// TIA Portal project "Project_farmas_1234_Before_trangsfer" (V14)

(* hardware
DEVICE "S7-1200 station_1"  S7-1200 Station
   slot 0: "Rack_0"  S7-1200 Rack  Rack  V1.0
   slot 1: "PLC_1"  CPU 1215C DC/DC/DC  6ES7 215-1AG40-0XB0  V4.2
   slot 2: "DI 8x24VDC/DQ 8xRelay_1"  SM 1223 DI8/DQ8 x relay  6ES7 223-1PH32-0XB0  V2.0
DEVICE "GSD device_1"  GSD.Device.PN
   slot 0: "Rack"  Rack  V1.0
   slot 0: "Input Universal Full"  Input Universal Full
   slot 0: "Output Universal Full"  Output Universal Full
   slot 0: "multicontrol11"  MultiControl PROFINET  1101834  2.??
      slot 0: "MultiControl DAP"  MultiControl DAP
      slot 1: "PROFINET Network Interface"  PROFINET Network Interface
         slot 1: "Port 1"  Port 1
         slot 2: "Port 2"  Port 2
      slot 1: "Process Image Input_1"  Process Image Input
      slot 2: "Access Point for acyclic Services_1"  Access Point for acyclic Services
         slot 0: "Access Point for acyclic Services"  Access Point for acyclic Services
      slot 3: "Process Image Output_1"  Process Image Output
DEVICE "GSD device_2"  GSD.Device.PN
   slot 0: "Rack"  Rack  V1.0
   slot 0: "Input Universal Full"  Input Universal Full
   slot 0: "Output Universal Full"  Output Universal Full
   slot 0: "multicontrol12"  MultiControl PROFINET  1101834  2.??
      slot 0: "MultiControl DAP"  MultiControl DAP
      slot 1: "PROFINET Network Interface"  PROFINET Network Interface
         slot 1: "Port 1"  Port 1
         slot 2: "Port 2"  Port 2
      slot 1: "Process Image Input_1"  Process Image Input
      slot 2: "Access Point for acyclic Services_1"  Access Point for acyclic Services
         slot 0: "Access Point for acyclic Services"  Access Point for acyclic Services
      slot 3: "Process Image Output_1"  Process Image Output
DEVICE "GSD device_3"  GSD.Device.PN
   slot 0: "Rack"  Rack  V1.0
   slot 0: "Input Universal Full"  Input Universal Full
   slot 0: "Output Universal Full"  Output Universal Full
   slot 0: "multicontrol13"  MultiControl PROFINET  1101834  2.??
      slot 0: "MultiControl DAP"  MultiControl DAP
      slot 1: "PROFINET Network Interface"  PROFINET Network Interface
         slot 1: "Port 1"  Port 1
         slot 2: "Port 2"  Port 2
      slot 1: "Process Image Input_1"  Process Image Input
      slot 2: "Access Point for acyclic Services_1"  Access Point for acyclic Services
         slot 0: "Access Point for acyclic Services"  Access Point for acyclic Services
      slot 3: "Process Image Output_1"  Process Image Output
DEVICE "GSD device_4"  GSD.Device.PN
   slot 0: "Rack"  Rack  V1.0
   slot 0: "Input Universal Full"  Input Universal Full
   slot 0: "Output Universal Full"  Output Universal Full
   slot 0: "multicontrol14"  MultiControl PROFINET  1101834  2.??
      slot 0: "MultiControl DAP"  MultiControl DAP
      slot 1: "PROFINET Network Interface"  PROFINET Network Interface
         slot 1: "Port 1"  Port 1
         slot 2: "Port 2"  Port 2
      slot 1: "Process Image Input_1"  Process Image Input
      slot 2: "Access Point for acyclic Services_1"  Access Point for acyclic Services
         slot 0: "Access Point for acyclic Services"  Access Point for acyclic Services
      slot 3: "Process Image Output_1"  Process Image Output
DEVICE "GSD device_5"  GSD.Device.PN
   slot 0: "Rack"  Rack  V1.0
   slot 0: "Input Universal Full"  Input Universal Full
   slot 0: "Output Universal Full"  Output Universal Full
   slot 0: "multicontrol15"  MultiControl PROFINET  1101834  2.??
      slot 0: "MultiControl DAP"  MultiControl DAP
      slot 1: "PROFINET Network Interface"  PROFINET Network Interface
         slot 1: "Port 1"  Port 1
         slot 2: "Port 2"  Port 2
      slot 1: "Process Image Input_1"  Process Image Input
      slot 2: "Access Point for acyclic Services_1"  Access Point for acyclic Services
         slot 0: "Access Point for acyclic Services"  Access Point for acyclic Services
      slot 3: "Process Image Output_1"  Process Image Output
DEVICE "GSD device_6"  GSD.Device.PN
   slot 0: "Rack"  Rack  V1.0
   slot 0: "Input Universal Full"  Input Universal Full
   slot 0: "Output Universal Full"  Output Universal Full
   slot 0: "multicontrol16"  MultiControl PROFINET  1101834  2.??
      slot 0: "MultiControl DAP"  MultiControl DAP
      slot 1: "PROFINET Network Interface"  PROFINET Network Interface
         slot 1: "Port 1"  Port 1
         slot 2: "Port 2"  Port 2
      slot 1: "Process Image Input_1"  Process Image Input
      slot 2: "Access Point for acyclic Services_1"  Access Point for acyclic Services
         slot 0: "Access Point for acyclic Services"  Access Point for acyclic Services
      slot 3: "Process Image Output_1"  Process Image Output
*)

// ===== PLC "PLC_1"  CPU 1215C DC/DC/DC =====

VAR_GLOBAL   // PLC tag table "Default tag table"
   "sensor_long_transfer" AT %I0.1 : Bool;
   "sensor_home_short_transfer" AT %I0.2 : Bool;
   "sensor_start_short_transfer" AT %I0.3 : Bool;
   "sensor_1_metal_pusher" AT %I0.6 : Bool;
   "sensor_2_metal_pusher" AT %I0.5 : Bool;
   "sensor_1_scale_pusher" AT %I1.0 : Bool;
   "sensor_2_scale_pusher" AT %I0.7 : Bool;
   "sensor_drive_control" AT %I2.0 : Bool;
   "start" AT %I0.4 : Bool;
   "sensor_5_13" AT %I2.1 : Bool;
   "13_sensor_1" AT %I140.0 : Bool;
   "13_sensor_2" AT %I140.1 : Bool;
   "13_sensor_3" AT %I140.2 : Bool;
   "13_sensor_4" AT %I140.3 : Bool;
   "14_sensor_1" AT %I176.0 : Bool;
   "14_sensor_2" AT %I176.1 : Bool;
   "14_sensor_3" AT %I176.2 : Bool;
   "14_sensor_4" AT %I176.3 : Bool;
   "15_sensor_1" AT %I212.0 : Bool;
   "15_sensor_2" AT %I212.1 : Bool;
   "15_sensor_3" AT %I212.2 : Bool;
   "15_sensor_4" AT %I212.3 : Bool;
   "16_sensor_1" AT %I248.0 : Bool;
   "16_sensor_2" AT %I248.1 : Bool;
   "16_sensor_3" AT %I248.2 : Bool;
   "16_sensor_4" AT %I248.3 : Bool;
   "signal_left" AT %I1.2 : Bool;
   "signal_right" AT %I1.3 : Bool;
   "signal_reject_scale" AT %I1.5 : Bool;
   "signal_good_bad" AT %I2.3 : Bool;
   "signal_reject_metal" AT %I1.1 : Bool;
   "signal_scale" AT %I2.2 : Bool;
   "Tag_12" AT %I1.4 : Bool;
   "Tag_134" AT %I2.5 : Bool;
   "Tag_174" AT %I2.4 : Bool;
   "Tag_227" AT %I2.7 : Bool;
   "Tag_228" AT %I2.6 : Bool;
   "Tag_274" AT %I0.0 : Bool;
   "pulse_step" AT %Q0.0 : Bool;
   "direction_step" AT %Q0.1 : Bool;
   "run_left_short_transfer" AT %Q0.3 : Bool;
   "run_right_short_transfer" AT %Q0.2 : Bool;
   "run_long_transfer" AT %Q0.4 : Bool;
   "valve_metal_pusher" AT %Q0.5 : Bool;
   "valve_scale_pusher" AT %Q0.6 : Bool;
   "valve_long_transfer" AT %Q0.7 : Bool;
   "speed_drive_control" AT %Q1.0 : Bool;
   "direction_drive_control" AT %Q1.1 : Bool;
   "run_lamp" AT %Q2.0 : Bool;
   "13_RD1" AT %QB89 : Byte;
   "13_RD2" AT %QB90 : Byte;
   "13_RD3" AT %QB91 : Byte;
   "13_RD4" AT %QB92 : Byte;
   "14_RD1" AT %QB99 : Byte;
   "14_RD2" AT %QB100 : Byte;
   "14_RD3" AT %QB101 : Byte;
   "14_RD4" AT %QB102 : Byte;
   "15_RD1" AT %QB109 : Byte;
   "15_RD3" AT %QB110 : Byte;
   "15_RD2" AT %QB111 : Byte;
   "15_RD4" AT %QB112 : Byte;
   "16_RD1" AT %QB119 : Byte;
   "16_RD2" AT %QB120 : Byte;
   "16_RD3" AT %QB121 : Byte;
   "16_RD4" AT %QB122 : Byte;
   "Tag_206" AT %Q2.4 : Bool;
   "Tag_223" AT %Q2.1 : Bool;
   "Tag_224" AT %Q2.2 : Bool;
   "Tag_225" AT %Q2.3 : Bool;
   "temp_left" AT %M0.0 : Bool;
   "temp_right" AT %M0.1 : Bool;
   "temp_up_down_short_transfer" AT %M0.2 : Bool;
   "temp_stop_long_transfer" AT %M0.3 : Bool;
   "temp_metal_pusher" AT %M1.1 : Bool;
   "temp_13_sensor_1" AT %M13.1 : Bool;
   "temp_13_sensor_2" AT %M13.2 : Bool;
   "temp_13_sensor_3" AT %M13.3 : Bool;
   "temp_13_sensor_4" AT %M13.4 : Bool;
   "temp_14_sensor_1" AT %M14.1 : Bool;
   "temp_14_sensor_2" AT %M14.2 : Bool;
   "temp_14_sensor_3" AT %M14.3 : Bool;
   "temp_14_sensor_4" AT %M14.4 : Bool;
   "temp_15_sensor_1" AT %M15.1 : Bool;
   "temp_15_sensor_2" AT %M15.2 : Bool;
   "temp_15_sensor_3" AT %M15.3 : Bool;
   "temp_15_sensor_4" AT %M15.4 : Bool;
   "temp_16_sensor_1" AT %M16.1 : Bool;
   "temp_16_sensor_2" AT %M16.2 : Bool;
   "temp_16_sensor_3" AT %M16.3 : Bool;
   "temp_16_sensor_4" AT %M16.4 : Bool;
   "temp_drive_control" AT %M17.0 : Bool;
   "temp_signal_good_bad" AT %M17.1 : Bool;
   "temp_reject_metal" AT %M17.2 : Bool;
   "temp_reject_scale" AT %M17.3 : Bool;
   "temp_scale_pusher" AT %M1.2 : Bool;
   "Tag_1" AT %M16.6 : Bool;
   "Tag_2" AT %M0.4 : Bool;
   "Tag_3" AT %M100.0 : Bool;
   "Tag_4" AT %M100.1 : Bool;
   "Tag_5" AT %M100.2 : Bool;
   "Tag_6" AT %M100.3 : Bool;
   "Tag_7" AT %M100.4 : Bool;
   "Tag_8" AT %M100.6 : Bool;
   "Tag_9" AT %M101.0 : Bool;
   "Tag_10" AT %M101.5 : Bool;
   "Tag_11" AT %M105.6 : Bool;
   "Tag_13" AT %M150.0 : Bool;
   "Tag_14" AT %M150.1 : Bool;
   "Tag_15" AT %M200.2 : Bool;
   "Tag_16" AT %M1000.0 : Bool;
   "Tag_17" AT %M200.1 : Bool;
   "Tag_18" AT %M1000.1 : Bool;
   "Tag_19" AT %M1000.2 : Bool;
   "Tag_20" AT %M200.7 : Bool;
   "Tag_21" AT %M200.0 : Bool;
   "Tag_22" AT %M201.1 : Bool;
   "Tag_23" AT %M151.0 : Bool;
   "Tag_24" AT %M151.1 : Bool;
   "Tag_25" AT %M201.7 : Bool;
   "Tag_26" AT %M149.0 : Bool;
   "Tag_27" AT %M149.1 : Bool;
   "Tag_28" AT %M199.7 : Bool;
   "Tag_29" AT %M199.0 : Bool;
   "Tag_30" AT %M199.1 : Bool;
   "Tag_31" AT %M999.0 : Bool;
   "Tag_32" AT %M999.1 : Bool;
   "Tag_33" AT %M999.2 : Bool;
   "Tag_34" AT %M199.2 : Bool;
   "Tag_35" AT %M202.1 : Bool;
   "Tag_36" AT %M201.0 : Bool;
   "Tag_37" AT %M201.2 : Bool;
   "Tag_38" AT %M1001.2 : Bool;
   "Tag_39" AT %M1001.1 : Bool;
   "Tag_40" AT %M1001.0 : Bool;
   "Tag_41" AT %M158.0 : Bool;
   "Tag_42" AT %M158.1 : Bool;
   "Tag_43" AT %M208.7 : Bool;
   "Tag_44" AT %M203.1 : Bool;
   "Tag_45" AT %M208.0 : Bool;
   "Tag_46" AT %M208.1 : Bool;
   "Tag_47" AT %M159.0 : Bool;
   "Tag_48" AT %M159.1 : Bool;
   "Tag_49" AT %M209.7 : Bool;
   "Tag_50" AT %M210.1 : Bool;
   "Tag_51" AT %M209.0 : Bool;
   "Tag_52" AT %M209.1 : Bool;
   "Tag_53" AT %M209.2 : Bool;
   "Tag_54" AT %M1009.0 : Bool;
   "Tag_55" AT %M1009.1 : Bool;
   "Tag_56" AT %M160.0 : Bool;
   "Tag_57" AT %M160.1 : Bool;
   "Tag_58" AT %M210.7 : Bool;
   "Tag_59" AT %M211.1 : Bool;
   "Tag_60" AT %M210.0 : Bool;
   "Tag_61" AT %M210.2 : Bool;
   "Tag_62" AT %M161.0 : Bool;
   "Tag_63" AT %M161.1 : Bool;
   "Tag_64" AT %M211.7 : Bool;
   "Tag_65" AT %M212.1 : Bool;
   "Tag_66" AT %M211.0 : Bool;
   "Tag_67" AT %M1010.0 : Bool;
   "Tag_68" AT %M1010.1 : Bool;
   "Tag_69" AT %M1010.2 : Bool;
   "Tag_70" AT %M211.2 : Bool;
   "Tag_71" AT %M1011.0 : Bool;
   "Tag_72" AT %M1011.1 : Bool;
   "Tag_73" AT %M1011.2 : Bool;
   "Tag_74" AT %M162.0 : Bool;
   "Tag_75" AT %M162.1 : Bool;
   "Tag_76" AT %M212.7 : Bool;
   "Tag_77" AT %M213.1 : Bool;
   "Tag_78" AT %M212.0 : Bool;
   "Tag_79" AT %M153.0 : Bool;
   "Tag_80" AT %M153.1 : Bool;
   "Tag_81" AT %M156.0 : Bool;
   "Tag_82" AT %M156.1 : Bool;
   "Tag_83" AT %M206.7 : Bool;
   "Tag_84" AT %M206.0 : Bool;
   "Tag_85" AT %M206.1 : Bool;
   "Tag_86" AT %M206.2 : Bool;
   "Tag_87" AT %M1006.0 : Bool;
   "Tag_88" AT %M1006.1 : Bool;
   "Tag_89" AT %M1006.2 : Bool;
   "Tag_90" AT %M152.0 : Bool;
   "Tag_91" AT %M152.1 : Bool;
   "Tag_92" AT %M202.7 : Bool;
   "Tag_93" AT %M202.0 : Bool;
   "Tag_94" AT %M202.2 : Bool;
   "Tag_95" AT %M203.3 : Bool;
   "Tag_96" AT %M1002.0 : Bool;
   "Tag_97" AT %M1002.1 : Bool;
   "Tag_98" AT %M1002.2 : Bool;
   "Tag_99" AT %M207.5 : Bool;
   "Tag_100" AT %M203.7 : Bool;
   "Tag_101" AT %M204.1 : Bool;
   "Tag_102" AT %M203.0 : Bool;
   "Tag_103" AT %M203.2 : Bool;
   "Tag_104" AT %M1003.2 : Bool;
   "Tag_105" AT %M203.4 : Bool;
   "Tag_106" AT %M204.5 : Bool;
   "Tag_107" AT %M1006.5 : Bool;
   "Tag_108" AT %M207.4 : Bool;
   "Tag_109" AT %M1006.6 : Bool;
   "Tag_110" AT %M1007.0 : Bool;
   "Tag_111" AT %M1007.1 : Bool;
   "Tag_112" AT %M1007.2 : Bool;
   "Tag_113" AT %M1007.4 : Bool;
   "Tag_114" AT %M1007.5 : Bool;
   "Tag_115" AT %M208.2 : Bool;
   "Tag_116" AT %M1008.0 : Bool;
   "Tag_117" AT %M1008.1 : Bool;
   "Tag_118" AT %M1008.2 : Bool;
   "Tag_119" AT %M147.0 : Bool;
   "Tag_120" AT %M1008.6 : Bool;
   "Tag_121" AT %M1008.7 : Bool;
   "Tag_122" AT %M198.0 : Bool;
   "Tag_123" AT %M300.7 : Bool;
   "Tag_124" AT %M212.2 : Bool;
   "Tag_125" AT %M1012.0 : Bool;
   "Tag_126" AT %M1012.1 : Bool;
   "Tag_127" AT %M1012.2 : Bool;
   "Tag_128" AT %M163.0 : Bool;
   "Tag_129" AT %M163.1 : Bool;
   "Tag_130" AT %M213.7 : Bool;
   "Tag_131" AT %M214.1 : Bool;
   "Tag_132" AT %M213.0 : Bool;
   "Tag_133" AT %M213.2 : Bool;
   "Tag_135" AT %M1001.3 : Bool;
   "Tag_136" AT %M1013.0 : Bool;
   "Tag_137" AT %M1013.3 : Bool;
   "Tag_138" AT %M1013.1 : Bool;
   "Tag_139" AT %M1013.2 : Bool;
   "Tag_140" AT %M164.0 : Bool;
   "Tag_141" AT %M164.1 : Bool;
   "Tag_142" AT %M214.7 : Bool;
   "Tag_143" AT %M215.1 : Bool;
   "Tag_144" AT %M214.0 : Bool;
   "Tag_145" AT %M217.0 : Bool;
   "Tag_146" AT %M214.2 : Bool;
   "Tag_147" AT %M1014.0 : Bool;
   "Tag_148" AT %M1014.1 : Bool;
   "Tag_149" AT %M1014.2 : Bool;
   "Tag_150" AT %M0.5 : Bool;
   "Tag_151" AT %M1020.0 : Bool;
   "Tag_152" AT %M1020.7 : Bool;
   "Tag_153" AT %M1021.0 : Bool;
   "Tag_154" AT %M1021.1 : Bool;
   "Tag_155" AT %M1022.2 : Bool;
   "Tag_156" AT %M146.1 : Bool;
   "Tag_157" AT %M146.0 : Bool;
   "Tag_158" AT %M1023.0 : Bool;
   "Tag_159" AT %M165.0 : Bool;
   "Tag_160" AT %M165.1 : Bool;
   "Tag_161" AT %M215.7 : Bool;
   "Tag_162" AT %M216.1 : Bool;
   "Tag_163" AT %M215.0 : Bool;
   "Tag_164" AT %M215.2 : Bool;
   "Tag_165" AT %M1015.0 : Bool;
   "Tag_166" AT %M214.3 : Bool;
   "Tag_167" AT %M1025.0 : Bool;
   "Tag_168" AT %M1025.1 : Bool;
   "Tag_169" AT %M166.0 : Bool;
   "Tag_170" AT %M166.1 : Bool;
   "Tag_171" AT %M216.7 : Bool;
   "Tag_172" AT %M217.1 : Bool;
   "Tag_173" AT %M216.0 : Bool;
   "Tag_175" AT %M216.2 : Bool;
   "Tag_176" AT %M1016.0 : Bool;
   "Tag_177" AT %M1016.1 : Bool;
   "Tag_178" AT %M1016.2 : Bool;
   "Tag_179" AT %MW10 : Word;
   "Tag_180" AT %M1023.2 : Bool;
   "Tag_181" AT %M1023.3 : Bool;
   "Tag_182" AT %M1024.0 : Bool;
   "Tag_183" AT %M1024.1 : Bool;
   "Tag_184" AT %M1024.4 : Bool;
   "Tag_185" AT %M170.0 : Bool;
   "System_Byte" AT %MB4095 : Byte;
   "FirstScan" AT %M4095.0 : Bool;
   "DiagStatusUpdate" AT %M4095.1 : Bool;
   "AlwaysTRUE" AT %M4095.2 : Bool;
   "AlwaysFALSE" AT %M4095.3 : Bool;
   "System_Byte(1)" AT %MB1 : Byte;
   "Tag_186" AT %M1026.4 : Bool;
   "Tag_187" AT %M1028.0 : Bool;
   "Tag_188" AT %M1027.0 : Bool;
   "Tag_189" AT %M1500.0 : Bool;
   "Tag_190" AT %M208.5 : Bool;
   "Tag_191" AT %M1036.5 : Bool;
   "Tag_192" AT %M1030.0 : Bool;
   "Tag_193" AT %M1030.1 : Bool;
   "Tag_194" AT %M1035.2 : Bool;
   "Tag_195" AT %M1035.3 : Bool;
   "Tag_196" AT %M1035.6 : Bool;
   "Tag_197" AT %M1036.0 : Bool;
   "Tag_198" AT %M1033.6 : Bool;
   "Tag_199" AT %M300.3 : Bool;
   "Tag_200" AT %M1044.0 : Bool;
   "Tag_201" AT %M300.2 : Bool;
   "Tag_202" AT %M1044.1 : Bool;
   "Tag_203" AT %M1040.0 : Bool;
   "Tag_204" AT %M1040.3 : Bool;
   "Tag_205" AT %M1047.0 : Bool;
   "Tag_207" AT %M400.0 : Bool;
   "Tag_208" AT %M400.1 : Bool;
   "Tag_209" AT %M399.0 : Bool;
   "Tag_210" AT %M400.5 : Bool;
   "Tag_211" AT %M400.6 : Bool;
   "Tag_212" AT %M400.7 : Bool;
   "Tag_213" AT %M800.0 : Bool;
   "Tag_214" AT %M800.3 : Bool;
   "Tag_215" AT %M801.0 : Bool;
   "Tag_216" AT %M401.1 : Bool;
   "Tag_217" AT %M801.1 : Bool;
   "Tag_218" AT %M401.2 : Bool;
   "Tag_219" AT %M801.2 : Bool;
   "Tag_220" AT %M1080.0 : Bool;
   "Tag_221" AT %M404.0 : Bool;
   "Tag_222" AT %M500.0 : Bool;
   "Tag_226" AT %M500.1 : Bool;
   "Clock_Byte" AT %MB410 : Byte;
   "Clock_10Hz" AT %M410.0 : Bool;
   "Clock_5Hz" AT %M410.1 : Bool;
   "Clock_2.5Hz" AT %M410.2 : Bool;
   "Clock_2Hz" AT %M410.3 : Bool;
   "Clock_1.25Hz" AT %M410.4 : Bool;
   "Clock_1Hz" AT %M410.5 : Bool;
   "Clock_0.625Hz" AT %M410.6 : Bool;
   "Clock_0.5Hz" AT %M410.7 : Bool;
   "Tag_229" AT %M420.0 : Bool;
   "Tag_230" AT %M500.2 : Bool;
   "Tag_231" AT %M420.1 : Bool;
   "Tag_232" AT %M500.3 : Bool;
   "Tag_233" AT %M500.4 : Bool;
   "Tag_234" AT %M400.4 : Bool;
   "Tag_235" AT %M420.4 : Bool;
   "Tag_236" AT %M500.7 : Bool;
   "Tag_237" AT %M1053.0 : Bool;
   "Tag_238" AT %M1053.1 : Bool;
   "Tag_239" AT %M1053.3 : Bool;
   "Tag_240" AT %M1070.0 : Bool;
   "Tag_241" AT %M700.0 : Bool;
   "Tag_242" AT %M489.0 : Bool;
   "Tag_243" AT %M500.5 : Bool;
   "Tag_244" AT %M500.6 : Bool;
   "Tag_245" AT %M1071.1 : Bool;
   "Tag_246" AT %M293.1 : Bool;
   "Tag_247" AT %M1071.2 : Bool;
   "Tag_248" AT %M1071.3 : Bool;
   "Tag_249" AT %M1071.4 : Bool;
   "Tag_250" AT %M1072.1 : Bool;
   "Tag_251" AT %M293.2 : Bool;
   "Tag_252" AT %M388.0 : Bool;
   "Tag_253" AT %M1077.2 : Bool;
   "Tag_254" AT %M2.6 : Bool;
   "Tag_255" AT %M1074.0 : Bool;
   "Tag_256" AT %M1075.0 : Bool;
   "Tag_257" AT %M183.0 : Bool;
   "Tag_258" AT %M1090.0 : Bool;
   "Tag_259" AT %M1090.1 : Bool;
   "Tag_260" AT %M1090.3 : Bool;
   "Tag_261" AT %M1090.4 : Bool;
   "Tag_262" AT %M1090.5 : Bool;
   "Tag_263" AT %M1090.6 : Bool;
   "Tag_264" AT %M1091.0 : Bool;
   "Tag_265" AT %M1091.1 : Bool;
   "Tag_266" AT %M1060.0 : Bool;
   "Tag_267" AT %M1060.1 : Bool;
   "Tag_268" AT %M1060.2 : Bool;
   "Tag_269" AT %M1060.3 : Bool;
   "Tag_270" AT %M1060.4 : Bool;
   "Tag_271" AT %M1060.5 : Bool;
   "Tag_272" AT %M1060.6 : Bool;
   "Tag_273" AT %M489.1 : Bool;
   "Tag_275" AT %M1061.0 : Bool;
   "Tag_276" AT %M489.2 : Bool;
   "Tag_277" AT %M489.4 : Bool;
   "Tag_278" AT %M1061.2 : Bool;
END_VAR

DATA_BLOCK "Connect_PC"   // DB1
{ S7_Optimized_Access := 'FALSE' }
VERSION : 0.1
   VAR
      Scan_check_metal : Byte := 0;
      weight_pusher : Byte := 0;
      print_pusher : Byte := 0;
      sensor_before_metal_scan : Byte := 0;
      metal_check_result : Byte := 0;
      sensor_after_metal_check : Byte := 0;
      metal_pusher : Byte := 0;
      sensor_tranfer : Byte := 0;
      sensor_left : Byte := 0;
      sensor_right : Byte := 0;
      EMG : Byte := 0;
   END_VAR
BEGIN
END_DATA_BLOCK

// folder: System blocks/Program resources

DATA_BLOCK "TZ7-1"   // DB6
{ S7_Optimized_Access := 'TRUE' }
AUTHOR : Simatic
FAMILY : IEC
NAME : IEC_TMR
VERSION : 1.0
// stored: InstanceOfName IEC_TIMER
"IEC_TIMER"
BEGIN
END_DATA_BLOCK

DATA_BLOCK "IEC_Timer_0_DB"   // DB7
{ S7_Optimized_Access := 'TRUE' }
AUTHOR : Simatic
FAMILY : IEC
NAME : IEC_TMR
VERSION : 1.0
// stored: InstanceOfName IEC_TIMER
"IEC_TIMER"
BEGIN
END_DATA_BLOCK

DATA_BLOCK "T13-1"   // DB8
{ S7_Optimized_Access := 'TRUE' }
AUTHOR : Simatic
FAMILY : IEC
NAME : IEC_TMR
VERSION : 1.0
// stored: InstanceOfName IEC_TIMER
"IEC_TIMER"
BEGIN
END_DATA_BLOCK

DATA_BLOCK "T13-2"   // DB9
{ S7_Optimized_Access := 'TRUE' }
AUTHOR : Simatic
FAMILY : IEC
NAME : IEC_TMR
VERSION : 1.0
// stored: InstanceOfName IEC_TIMER
"IEC_TIMER"
BEGIN
END_DATA_BLOCK

DATA_BLOCK "IEC_Timer_0_DB_9"   // DB10
{ S7_Optimized_Access := 'TRUE' }
AUTHOR : Simatic
FAMILY : IEC
NAME : IEC_TMR
VERSION : 1.0
// stored: InstanceOfName IEC_TIMER
"IEC_TIMER"
BEGIN
END_DATA_BLOCK

DATA_BLOCK "T9-1"   // DB11
{ S7_Optimized_Access := 'TRUE' }
AUTHOR : Simatic
FAMILY : IEC
NAME : IEC_TMR
VERSION : 1.0
// stored: InstanceOfName IEC_TIMER
"IEC_TIMER"
BEGIN
END_DATA_BLOCK

DATA_BLOCK "IEC_Timer_0_DB_1"   // DB12
{ S7_Optimized_Access := 'TRUE' }
AUTHOR : Simatic
FAMILY : IEC
NAME : IEC_TMR
VERSION : 1.0
// stored: InstanceOfName IEC_TIMER
"IEC_TIMER"
BEGIN
END_DATA_BLOCK

DATA_BLOCK "IEC_Timer_0_DB_2"   // DB13
{ S7_Optimized_Access := 'TRUE' }
AUTHOR : Simatic
FAMILY : IEC
NAME : IEC_TMR
VERSION : 1.0
// stored: InstanceOfName IEC_TIMER
"IEC_TIMER"
BEGIN
END_DATA_BLOCK

DATA_BLOCK "IEC_Timer_0_DB_3"   // DB14
{ S7_Optimized_Access := 'TRUE' }
AUTHOR : Simatic
FAMILY : IEC
NAME : IEC_TMR
VERSION : 1.0
// stored: InstanceOfName IEC_TIMER
"IEC_TIMER"
BEGIN
END_DATA_BLOCK

DATA_BLOCK "IEC_Timer_0_DB_4"   // DB15
{ S7_Optimized_Access := 'TRUE' }
AUTHOR : Simatic
FAMILY : IEC
NAME : IEC_TMR
VERSION : 1.0
// stored: InstanceOfName IEC_TIMER
"IEC_TIMER"
BEGIN
END_DATA_BLOCK

DATA_BLOCK "TZ12-1"   // DB16
{ S7_Optimized_Access := 'TRUE' }
AUTHOR : Simatic
FAMILY : IEC
NAME : IEC_TMR
VERSION : 1.0
// stored: InstanceOfName IEC_TIMER
"IEC_TIMER"
BEGIN
END_DATA_BLOCK

DATA_BLOCK "T3-1"   // DB17
{ S7_Optimized_Access := 'TRUE' }
AUTHOR : Simatic
FAMILY : IEC
NAME : IEC_TMR
VERSION : 1.0
// stored: InstanceOfName IEC_TIMER
"IEC_TIMER"
BEGIN
END_DATA_BLOCK

DATA_BLOCK "TZ3-1"   // DB18
{ S7_Optimized_Access := 'TRUE' }
AUTHOR : Simatic
FAMILY : IEC
NAME : IEC_TMR
VERSION : 1.0
// stored: InstanceOfName IEC_TIMER
"IEC_TIMER"
BEGIN
END_DATA_BLOCK

DATA_BLOCK "TZ3-2"   // DB19
{ S7_Optimized_Access := 'TRUE' }
AUTHOR : Simatic
FAMILY : IEC
NAME : IEC_TMR
VERSION : 1.0
// stored: InstanceOfName IEC_TIMER
"IEC_TIMER"
BEGIN
END_DATA_BLOCK

DATA_BLOCK "TZ5-2"   // DB20
{ S7_Optimized_Access := 'TRUE' }
AUTHOR : Simatic
FAMILY : IEC
NAME : IEC_TMR
VERSION : 1.0
// stored: InstanceOfName IEC_TIMER
"IEC_TIMER"
BEGIN
END_DATA_BLOCK

DATA_BLOCK "TZ5-1"   // DB21
{ S7_Optimized_Access := 'TRUE' }
AUTHOR : Simatic
FAMILY : IEC
NAME : IEC_TMR
VERSION : 1.0
// stored: InstanceOfName IEC_TIMER
"IEC_TIMER"
BEGIN
END_DATA_BLOCK

DATA_BLOCK "T5-1"   // DB22
{ S7_Optimized_Access := 'TRUE' }
AUTHOR : Simatic
FAMILY : IEC
NAME : IEC_TMR
VERSION : 1.0
// stored: InstanceOfName IEC_TIMER
"IEC_TIMER"
BEGIN
END_DATA_BLOCK

DATA_BLOCK "T5-2"   // DB23
{ S7_Optimized_Access := 'TRUE' }
AUTHOR : Simatic
FAMILY : IEC
NAME : IEC_TMR
VERSION : 1.0
// stored: InstanceOfName IEC_TIMER
"IEC_TIMER"
BEGIN
END_DATA_BLOCK

DATA_BLOCK "T9-2"   // DB24
{ S7_Optimized_Access := 'TRUE' }
AUTHOR : Simatic
FAMILY : IEC
NAME : IEC_TMR
VERSION : 1.0
// stored: InstanceOfName IEC_TIMER
"IEC_TIMER"
BEGIN
END_DATA_BLOCK

DATA_BLOCK "T10-1"   // DB25
{ S7_Optimized_Access := 'TRUE' }
AUTHOR : Simatic
FAMILY : IEC
NAME : IEC_TMR
VERSION : 1.0
// stored: InstanceOfName IEC_TIMER
"IEC_TIMER"
BEGIN
END_DATA_BLOCK

DATA_BLOCK "T10-2"   // DB26
{ S7_Optimized_Access := 'TRUE' }
AUTHOR : Simatic
FAMILY : IEC
NAME : IEC_TMR
VERSION : 1.0
// stored: InstanceOfName IEC_TIMER
"IEC_TIMER"
BEGIN
END_DATA_BLOCK

DATA_BLOCK "TZ10-1"   // DB27
{ S7_Optimized_Access := 'TRUE' }
AUTHOR : Simatic
FAMILY : IEC
NAME : IEC_TMR
VERSION : 1.0
// stored: InstanceOfName IEC_TIMER
"IEC_TIMER"
BEGIN
END_DATA_BLOCK

DATA_BLOCK "TZ10-2"   // DB28
{ S7_Optimized_Access := 'TRUE' }
AUTHOR : Simatic
FAMILY : IEC
NAME : IEC_TMR
VERSION : 1.0
// stored: InstanceOfName IEC_TIMER
"IEC_TIMER"
BEGIN
END_DATA_BLOCK

DATA_BLOCK "TZ9-2"   // DB29
{ S7_Optimized_Access := 'TRUE' }
AUTHOR : Simatic
FAMILY : IEC
NAME : IEC_TMR
VERSION : 1.0
// stored: InstanceOfName IEC_TIMER
"IEC_TIMER"
BEGIN
END_DATA_BLOCK

DATA_BLOCK "TZ9-1"   // DB30
{ S7_Optimized_Access := 'TRUE' }
AUTHOR : Simatic
FAMILY : IEC
NAME : IEC_TMR
VERSION : 1.0
// stored: InstanceOfName IEC_TIMER
"IEC_TIMER"
BEGIN
END_DATA_BLOCK

DATA_BLOCK "TZ11-2"   // DB31
{ S7_Optimized_Access := 'TRUE' }
AUTHOR : Simatic
FAMILY : IEC
NAME : IEC_TMR
VERSION : 1.0
// stored: InstanceOfName IEC_TIMER
"IEC_TIMER"
BEGIN
END_DATA_BLOCK

DATA_BLOCK "TZ11-1"   // DB32
{ S7_Optimized_Access := 'TRUE' }
AUTHOR : Simatic
FAMILY : IEC
NAME : IEC_TMR
VERSION : 1.0
// stored: InstanceOfName IEC_TIMER
"IEC_TIMER"
BEGIN
END_DATA_BLOCK

DATA_BLOCK "T11-1"   // DB33
{ S7_Optimized_Access := 'TRUE' }
AUTHOR : Simatic
FAMILY : IEC
NAME : IEC_TMR
VERSION : 1.0
// stored: InstanceOfName IEC_TIMER
"IEC_TIMER"
BEGIN
END_DATA_BLOCK

DATA_BLOCK "T11-2"   // DB34
{ S7_Optimized_Access := 'TRUE' }
AUTHOR : Simatic
FAMILY : IEC
NAME : IEC_TMR
VERSION : 1.0
// stored: InstanceOfName IEC_TIMER
"IEC_TIMER"
BEGIN
END_DATA_BLOCK

DATA_BLOCK "T12-1"   // DB35
{ S7_Optimized_Access := 'TRUE' }
AUTHOR : Simatic
FAMILY : IEC
NAME : IEC_TMR
VERSION : 1.0
// stored: InstanceOfName IEC_TIMER
"IEC_TIMER"
BEGIN
END_DATA_BLOCK

DATA_BLOCK "T12-2"   // DB36
{ S7_Optimized_Access := 'TRUE' }
AUTHOR : Simatic
FAMILY : IEC
NAME : IEC_TMR
VERSION : 1.0
// stored: InstanceOfName IEC_TIMER
"IEC_TIMER"
BEGIN
END_DATA_BLOCK

DATA_BLOCK "TZ2-1"   // DB37
{ S7_Optimized_Access := 'TRUE' }
AUTHOR : Simatic
FAMILY : IEC
NAME : IEC_TMR
VERSION : 1.0
// stored: InstanceOfName IEC_TIMER
"IEC_TIMER"
BEGIN
END_DATA_BLOCK

DATA_BLOCK "TZ2-2"   // DB38
{ S7_Optimized_Access := 'TRUE' }
AUTHOR : Simatic
FAMILY : IEC
NAME : IEC_TMR
VERSION : 1.0
// stored: InstanceOfName IEC_TIMER
"IEC_TIMER"
BEGIN
END_DATA_BLOCK

DATA_BLOCK "T2-1"   // DB39
{ S7_Optimized_Access := 'TRUE' }
AUTHOR : Simatic
FAMILY : IEC
NAME : IEC_TMR
VERSION : 1.0
// stored: InstanceOfName IEC_TIMER
"IEC_TIMER"
BEGIN
END_DATA_BLOCK

DATA_BLOCK "T2-2"   // DB40
{ S7_Optimized_Access := 'TRUE' }
AUTHOR : Simatic
FAMILY : IEC
NAME : IEC_TMR
VERSION : 1.0
// stored: InstanceOfName IEC_TIMER
"IEC_TIMER"
BEGIN
END_DATA_BLOCK

DATA_BLOCK "T3-2"   // DB41
{ S7_Optimized_Access := 'TRUE' }
AUTHOR : Simatic
FAMILY : IEC
NAME : IEC_TMR
VERSION : 1.0
// stored: InstanceOfName IEC_TIMER
"IEC_TIMER"
BEGIN
END_DATA_BLOCK

DATA_BLOCK "TZ12-2"   // DB42
{ S7_Optimized_Access := 'TRUE' }
AUTHOR : Simatic
FAMILY : IEC
NAME : IEC_TMR
VERSION : 1.0
// stored: InstanceOfName IEC_TIMER
"IEC_TIMER"
BEGIN
END_DATA_BLOCK

DATA_BLOCK "T6-1"   // DB43
{ S7_Optimized_Access := 'TRUE' }
AUTHOR : Simatic
FAMILY : IEC
NAME : IEC_TMR
VERSION : 1.0
// stored: InstanceOfName IEC_TIMER
"IEC_TIMER"
BEGIN
END_DATA_BLOCK

DATA_BLOCK "TZ13-1"   // DB44
{ S7_Optimized_Access := 'TRUE' }
AUTHOR : Simatic
FAMILY : IEC
NAME : IEC_TMR
VERSION : 1.0
// stored: InstanceOfName IEC_TIMER
"IEC_TIMER"
BEGIN
END_DATA_BLOCK

DATA_BLOCK "TZ6-1"   // DB45
{ S7_Optimized_Access := 'TRUE' }
AUTHOR : Simatic
FAMILY : IEC
NAME : IEC_TMR
VERSION : 1.0
// stored: InstanceOfName IEC_TIMER
"IEC_TIMER"
BEGIN
END_DATA_BLOCK

DATA_BLOCK "TZ6-2"   // DB46
{ S7_Optimized_Access := 'TRUE' }
AUTHOR : Simatic
FAMILY : IEC
NAME : IEC_TMR
VERSION : 1.0
// stored: InstanceOfName IEC_TIMER
"IEC_TIMER"
BEGIN
END_DATA_BLOCK

DATA_BLOCK "T6-2"   // DB47
{ S7_Optimized_Access := 'TRUE' }
AUTHOR : Simatic
FAMILY : IEC
NAME : IEC_TMR
VERSION : 1.0
// stored: InstanceOfName IEC_TIMER
"IEC_TIMER"
BEGIN
END_DATA_BLOCK

DATA_BLOCK "TZ13-2"   // DB48
{ S7_Optimized_Access := 'TRUE' }
AUTHOR : Simatic
FAMILY : IEC
NAME : IEC_TMR
VERSION : 1.0
// stored: InstanceOfName IEC_TIMER
"IEC_TIMER"
BEGIN
END_DATA_BLOCK

DATA_BLOCK "T-metal"   // DB49
{ S7_Optimized_Access := 'TRUE' }
AUTHOR : Simatic
FAMILY : IEC
NAME : IEC_TMR
VERSION : 1.0
// stored: InstanceOfName IEC_TIMER
"IEC_TIMER"
BEGIN
END_DATA_BLOCK

DATA_BLOCK "T7-2"   // DB50
{ S7_Optimized_Access := 'TRUE' }
AUTHOR : Simatic
FAMILY : IEC
NAME : IEC_TMR
VERSION : 1.0
// stored: InstanceOfName IEC_TIMER
"IEC_TIMER"
BEGIN
END_DATA_BLOCK

DATA_BLOCK "TZ7-2"   // DB51
{ S7_Optimized_Access := 'TRUE' }
AUTHOR : Simatic
FAMILY : IEC
NAME : IEC_TMR
VERSION : 1.0
// stored: InstanceOfName IEC_TIMER
"IEC_TIMER"
BEGIN
END_DATA_BLOCK

DATA_BLOCK "TZ7-3"   // DB52
{ S7_Optimized_Access := 'TRUE' }
AUTHOR : Simatic
FAMILY : IEC
NAME : IEC_TMR
VERSION : 1.0
// stored: InstanceOfName IEC_TIMER
"IEC_TIMER"
BEGIN
END_DATA_BLOCK

DATA_BLOCK "TM207"   // DB53
{ S7_Optimized_Access := 'TRUE' }
AUTHOR : Simatic
FAMILY : IEC
NAME : IEC_TMR
VERSION : 1.0
// stored: InstanceOfName IEC_TIMER
"IEC_TIMER"
BEGIN
END_DATA_BLOCK

DATA_BLOCK "IEC_Timer_0_DB_5"   // DB54
{ S7_Optimized_Access := 'TRUE' }
AUTHOR : Simatic
FAMILY : IEC
NAME : IEC_TMR
VERSION : 1.0
// stored: InstanceOfName IEC_TIMER
"IEC_TIMER"
BEGIN
END_DATA_BLOCK

DATA_BLOCK "TZ8-1"   // DB55
{ S7_Optimized_Access := 'TRUE' }
AUTHOR : Simatic
FAMILY : IEC
NAME : IEC_TMR
VERSION : 1.0
// stored: InstanceOfName IEC_TIMER
"IEC_TIMER"
BEGIN
END_DATA_BLOCK

DATA_BLOCK "TZ8-2"   // DB56
{ S7_Optimized_Access := 'TRUE' }
AUTHOR : Simatic
FAMILY : IEC
NAME : IEC_TMR
VERSION : 1.0
// stored: InstanceOfName IEC_TIMER
"IEC_TIMER"
BEGIN
END_DATA_BLOCK

DATA_BLOCK "T8-1"   // DB57
{ S7_Optimized_Access := 'TRUE' }
AUTHOR : Simatic
FAMILY : IEC
NAME : IEC_TMR
VERSION : 1.0
// stored: InstanceOfName IEC_TIMER
"IEC_TIMER"
BEGIN
END_DATA_BLOCK

DATA_BLOCK "T8-2"   // DB58
{ S7_Optimized_Access := 'TRUE' }
AUTHOR : Simatic
FAMILY : IEC
NAME : IEC_TMR
VERSION : 1.0
// stored: InstanceOfName IEC_TIMER
"IEC_TIMER"
BEGIN
END_DATA_BLOCK

DATA_BLOCK "TZ14-2"   // DB59
{ S7_Optimized_Access := 'TRUE' }
AUTHOR : Simatic
FAMILY : IEC
NAME : IEC_TMR
VERSION : 1.0
// stored: InstanceOfName IEC_TIMER
"IEC_TIMER"
BEGIN
END_DATA_BLOCK

DATA_BLOCK "TZ14-1"   // DB60
{ S7_Optimized_Access := 'TRUE' }
AUTHOR : Simatic
FAMILY : IEC
NAME : IEC_TMR
VERSION : 1.0
// stored: InstanceOfName IEC_TIMER
"IEC_TIMER"
BEGIN
END_DATA_BLOCK

DATA_BLOCK "T14-1"   // DB61
{ S7_Optimized_Access := 'TRUE' }
AUTHOR : Simatic
FAMILY : IEC
NAME : IEC_TMR
VERSION : 1.0
// stored: InstanceOfName IEC_TIMER
"IEC_TIMER"
BEGIN
END_DATA_BLOCK

DATA_BLOCK "T14-2"   // DB62
{ S7_Optimized_Access := 'TRUE' }
AUTHOR : Simatic
FAMILY : IEC
NAME : IEC_TMR
VERSION : 1.0
// stored: InstanceOfName IEC_TIMER
"IEC_TIMER"
BEGIN
END_DATA_BLOCK

DATA_BLOCK "T-SCALE"   // DB63
{ S7_Optimized_Access := 'TRUE' }
AUTHOR : Simatic
FAMILY : IEC
NAME : IEC_TMR
VERSION : 1.0
// stored: InstanceOfName IEC_TIMER
"IEC_TIMER"
BEGIN
END_DATA_BLOCK

DATA_BLOCK "IEC_Timer_0_DB_7"   // DB64
{ S7_Optimized_Access := 'TRUE' }
AUTHOR : Simatic
FAMILY : IEC
NAME : IEC_TMR
VERSION : 1.0
// stored: InstanceOfName IEC_TIMER
"IEC_TIMER"
BEGIN
END_DATA_BLOCK

DATA_BLOCK "IEC_Timer_0_DB_8"   // DB65
{ S7_Optimized_Access := 'TRUE' }
AUTHOR : Simatic
FAMILY : IEC
NAME : IEC_TMR
VERSION : 1.0
// stored: InstanceOfName IEC_TIMER
"IEC_TIMER"
BEGIN
END_DATA_BLOCK

DATA_BLOCK "TZ15-1"   // DB66
{ S7_Optimized_Access := 'TRUE' }
AUTHOR : Simatic
FAMILY : IEC
NAME : IEC_TMR
VERSION : 1.0
// stored: InstanceOfName IEC_TIMER
"IEC_TIMER"
BEGIN
END_DATA_BLOCK

DATA_BLOCK "TZ15-2"   // DB67
{ S7_Optimized_Access := 'TRUE' }
AUTHOR : Simatic
FAMILY : IEC
NAME : IEC_TMR
VERSION : 1.0
// stored: InstanceOfName IEC_TIMER
"IEC_TIMER"
BEGIN
END_DATA_BLOCK

DATA_BLOCK "T15-1"   // DB68
{ S7_Optimized_Access := 'TRUE' }
AUTHOR : Simatic
FAMILY : IEC
NAME : IEC_TMR
VERSION : 1.0
// stored: InstanceOfName IEC_TIMER
"IEC_TIMER"
BEGIN
END_DATA_BLOCK

DATA_BLOCK "T15-2"   // DB69
{ S7_Optimized_Access := 'TRUE' }
AUTHOR : Simatic
FAMILY : IEC
NAME : IEC_TMR
VERSION : 1.0
// stored: InstanceOfName IEC_TIMER
"IEC_TIMER"
BEGIN
END_DATA_BLOCK

DATA_BLOCK "T16-1"   // DB70
{ S7_Optimized_Access := 'TRUE' }
AUTHOR : Simatic
FAMILY : IEC
NAME : IEC_TMR
VERSION : 1.0
// stored: InstanceOfName IEC_TIMER
"IEC_TIMER"
BEGIN
END_DATA_BLOCK

DATA_BLOCK "T16-2"   // DB71
{ S7_Optimized_Access := 'TRUE' }
AUTHOR : Simatic
FAMILY : IEC
NAME : IEC_TMR
VERSION : 1.0
// stored: InstanceOfName IEC_TIMER
"IEC_TIMER"
BEGIN
END_DATA_BLOCK

DATA_BLOCK "TZ16-1"   // DB72
{ S7_Optimized_Access := 'TRUE' }
AUTHOR : Simatic
FAMILY : IEC
NAME : IEC_TMR
VERSION : 1.0
// stored: InstanceOfName IEC_TIMER
"IEC_TIMER"
BEGIN
END_DATA_BLOCK

DATA_BLOCK "TZ16-2"   // DB73
{ S7_Optimized_Access := 'TRUE' }
AUTHOR : Simatic
FAMILY : IEC
NAME : IEC_TMR
VERSION : 1.0
// stored: InstanceOfName IEC_TIMER
"IEC_TIMER"
BEGIN
END_DATA_BLOCK

DATA_BLOCK "TZ16-3"   // DB74
{ S7_Optimized_Access := 'TRUE' }
AUTHOR : Simatic
FAMILY : IEC
NAME : IEC_TMR
VERSION : 1.0
// stored: InstanceOfName IEC_TIMER
"IEC_TIMER"
BEGIN
END_DATA_BLOCK

DATA_BLOCK "IEC_Timer_0_DB_10"   // DB75
{ S7_Optimized_Access := 'TRUE' }
AUTHOR : Simatic
FAMILY : IEC
NAME : IEC_TMR
VERSION : 1.0
// stored: InstanceOfName IEC_TIMER
"IEC_TIMER"
BEGIN
END_DATA_BLOCK

DATA_BLOCK "T2-0"   // DB76
{ S7_Optimized_Access := 'TRUE' }
AUTHOR : Simatic
FAMILY : IEC
NAME : IEC_TMR
VERSION : 1.0
// stored: InstanceOfName IEC_TIMER
"IEC_TIMER"
BEGIN
END_DATA_BLOCK

DATA_BLOCK "IEC_Timer_0_DB_6"   // DB77
{ S7_Optimized_Access := 'TRUE' }
AUTHOR : Simatic
FAMILY : IEC
NAME : IEC_TMR
VERSION : 1.0
// stored: InstanceOfName IEC_TIMER
"IEC_TIMER"
BEGIN
END_DATA_BLOCK

DATA_BLOCK "IEC_Timer_0_DB_11"   // DB78
{ S7_Optimized_Access := 'TRUE' }
AUTHOR : Simatic
FAMILY : IEC
NAME : IEC_TMR
VERSION : 1.0
// stored: InstanceOfName IEC_TIMER
"IEC_TIMER"
BEGIN
END_DATA_BLOCK

DATA_BLOCK "tm208"   // DB79
{ S7_Optimized_Access := 'TRUE' }
AUTHOR : Simatic
FAMILY : IEC
NAME : IEC_TMR
VERSION : 1.0
// stored: InstanceOfName IEC_TIMER
"IEC_TIMER"
BEGIN
END_DATA_BLOCK

DATA_BLOCK "IEC_Timer_0_DB_12"   // DB80
{ S7_Optimized_Access := 'TRUE' }
AUTHOR : Simatic
FAMILY : IEC
NAME : IEC_TMR
VERSION : 1.0
// stored: InstanceOfName IEC_TIMER
"IEC_TIMER"
BEGIN
END_DATA_BLOCK

DATA_BLOCK "IEC_Timer_0_DB_13"   // DB81
{ S7_Optimized_Access := 'TRUE' }
AUTHOR : Simatic
FAMILY : IEC
NAME : IEC_TMR
VERSION : 1.0
// stored: InstanceOfName IEC_TIMER
"IEC_TIMER"
BEGIN
END_DATA_BLOCK

DATA_BLOCK "IEC_Timer_0_DB_14"   // DB82
{ S7_Optimized_Access := 'TRUE' }
AUTHOR : Simatic
FAMILY : IEC
NAME : IEC_TMR
VERSION : 1.0
// stored: InstanceOfName IEC_TIMER
"IEC_TIMER"
BEGIN
END_DATA_BLOCK

DATA_BLOCK "IEC_Timer_0_DB_15"   // DB83
{ S7_Optimized_Access := 'TRUE' }
AUTHOR : Simatic
FAMILY : IEC
NAME : IEC_TMR
VERSION : 1.0
// stored: InstanceOfName IEC_TIMER
"IEC_TIMER"
BEGIN
END_DATA_BLOCK

DATA_BLOCK "IEC_Timer_0_DB_16"   // DB84
{ S7_Optimized_Access := 'TRUE' }
AUTHOR : Simatic
FAMILY : IEC
NAME : IEC_TMR
VERSION : 1.0
// stored: InstanceOfName IEC_TIMER
"IEC_TIMER"
BEGIN
END_DATA_BLOCK

DATA_BLOCK "T_Error"   // DB85
{ S7_Optimized_Access := 'TRUE' }
AUTHOR : Simatic
FAMILY : IEC
NAME : IEC_TMR
VERSION : 1.0
// stored: InstanceOfName IEC_TIMER
"IEC_TIMER"
BEGIN
END_DATA_BLOCK

DATA_BLOCK "IEC_Timer_0_DB_18"   // DB86
{ S7_Optimized_Access := 'TRUE' }
AUTHOR : Simatic
FAMILY : IEC
NAME : IEC_TMR
VERSION : 1.0
// stored: InstanceOfName IEC_TIMER
"IEC_TIMER"
BEGIN
END_DATA_BLOCK

DATA_BLOCK "TPUSH"   // DB87
{ S7_Optimized_Access := 'TRUE' }
AUTHOR : Simatic
FAMILY : IEC
NAME : IEC_TMR
VERSION : 1.0
// stored: InstanceOfName IEC_TIMER
"IEC_TIMER"
BEGIN
END_DATA_BLOCK

DATA_BLOCK "T_METAL"   // DB88
{ S7_Optimized_Access := 'TRUE' }
AUTHOR : Simatic
FAMILY : IEC
NAME : IEC_TMR
VERSION : 1.0
// stored: InstanceOfName IEC_TIMER
"IEC_TIMER"
BEGIN
END_DATA_BLOCK

DATA_BLOCK "T_rr"   // DB89
{ S7_Optimized_Access := 'TRUE' }
AUTHOR : Simatic
FAMILY : IEC
NAME : IEC_TMR
VERSION : 1.0
// stored: InstanceOfName IEC_TIMER
"IEC_TIMER"
BEGIN
END_DATA_BLOCK

DATA_BLOCK "TR"   // DB90
{ S7_Optimized_Access := 'TRUE' }
AUTHOR : Simatic
FAMILY : IEC
NAME : IEC_TMR
VERSION : 1.0
// stored: InstanceOfName IEC_TIMER
"IEC_TIMER"
BEGIN
END_DATA_BLOCK

DATA_BLOCK "TR1"   // DB91
{ S7_Optimized_Access := 'TRUE' }
AUTHOR : Simatic
FAMILY : IEC
NAME : IEC_TMR
VERSION : 1.0
// stored: InstanceOfName IEC_TIMER
"IEC_TIMER"
BEGIN
END_DATA_BLOCK

DATA_BLOCK "TR2"   // DB92
{ S7_Optimized_Access := 'TRUE' }
AUTHOR : Simatic
FAMILY : IEC
NAME : IEC_TMR
VERSION : 1.0
// stored: InstanceOfName IEC_TIMER
"IEC_TIMER"
BEGIN
END_DATA_BLOCK

DATA_BLOCK "IEC_Timer_0_DB_17"   // DB93
{ S7_Optimized_Access := 'TRUE' }
AUTHOR : Simatic
FAMILY : IEC
NAME : IEC_TMR
VERSION : 1.0
// stored: InstanceOfName IEC_TIMER
"IEC_TIMER"
BEGIN
END_DATA_BLOCK

DATA_BLOCK "TM500"   // DB94
{ S7_Optimized_Access := 'TRUE' }
AUTHOR : Simatic
FAMILY : IEC
NAME : IEC_TMR
VERSION : 1.0
// stored: InstanceOfName IEC_TIMER
"IEC_TIMER"
BEGIN
END_DATA_BLOCK

DATA_BLOCK "IEC_Timer_0_DB_19"   // DB95
{ S7_Optimized_Access := 'TRUE' }
AUTHOR : Simatic
FAMILY : IEC
NAME : IEC_TMR
VERSION : 1.0
// stored: InstanceOfName IEC_TIMER
"IEC_TIMER"
BEGIN
END_DATA_BLOCK

DATA_BLOCK "IEC_Timer_0_DB_20"   // DB96
{ S7_Optimized_Access := 'TRUE' }
AUTHOR : Simatic
FAMILY : IEC
NAME : IEC_TMR
VERSION : 1.0
// stored: InstanceOfName IEC_TIMER
"IEC_TIMER"
BEGIN
END_DATA_BLOCK

DATA_BLOCK "IEC_Timer_0_DB_21"   // DB97
{ S7_Optimized_Access := 'TRUE' }
AUTHOR : Simatic
FAMILY : IEC
NAME : IEC_TMR
VERSION : 1.0
// stored: InstanceOfName IEC_TIMER
"IEC_TIMER"
BEGIN
END_DATA_BLOCK

DATA_BLOCK "T489.1"   // DB98
{ S7_Optimized_Access := 'TRUE' }
AUTHOR : Simatic
FAMILY : IEC
NAME : IEC_TMR
VERSION : 1.0
// stored: InstanceOfName IEC_TIMER
"IEC_TIMER"
BEGIN
END_DATA_BLOCK

DATA_BLOCK "IEC_Timer_0_DB_22"   // DB99
{ S7_Optimized_Access := 'TRUE' }
AUTHOR : Simatic
FAMILY : IEC
NAME : IEC_TMR
VERSION : 1.0
// stored: InstanceOfName IEC_TIMER
"IEC_TIMER"
BEGIN
END_DATA_BLOCK

DATA_BLOCK "IEC_Timer_0_DB_23"   // DB100
{ S7_Optimized_Access := 'TRUE' }
AUTHOR : Simatic
FAMILY : IEC
NAME : IEC_TMR
VERSION : 1.0
// stored: InstanceOfName IEC_TIMER
"IEC_TIMER"
BEGIN
END_DATA_BLOCK

DATA_BLOCK "IEC_Timer_0_DB_24"   // DB101
{ S7_Optimized_Access := 'TRUE' }
AUTHOR : Simatic
FAMILY : IEC
NAME : IEC_TMR
VERSION : 1.0
// stored: InstanceOfName IEC_TIMER
"IEC_TIMER"
BEGIN
END_DATA_BLOCK

// folder: (top level)

DATA_BLOCK "Axis_1"   // DB2, Motion_DB
{ S7_Optimized_Access := 'TRUE' }
AUTHOR : SIMATIC
FAMILY : BasicMC
NAME : TO_PosAx
VERSION : 6.0
// stored: InstanceOfName TO_PositioningAxis
"TO_PositioningAxis"
BEGIN
   // Axis.DirectionOutputEnabledCU = TRUE
   // Axis.OnlinePtoModeCUEnumValue = PTO (pulse A and direction B)
   // Axis.OnlinePtoModeCU = 16#0000_0002
   // Axis.SelectedChannel2EnumCU = %Q0.1
   // Axis.SelectedChannel1EnumCU = %Q0.0
   // Pulse.MinDeltaDeltaFrequencyCU = 0.004
   // Pulse.MaxDeltaDeltaFrequencyCU = 1.0E+10
   // Pulse.MinDeltaFrequencyCU = 0.005
   // Pulse.MaxDeltaFrequencyCU = 9.5E+9
   // Pulse.MinFrequencyCU = 1.0
   // Pulse.MaxFrequencyCU = 100000.0
   // Pulse.OutputSourceCU = 16#0000_0000
   // Axis.SelectPTO = 0
   // Axis.LengthUnit.LastDistance = -1
END_DATA_BLOCK

FUNCTION "transfer" : Void   // FC1, LAD
{ S7_Optimized_Access := 'TRUE' }
VERSION : 0.1
   VAR_TEMP   // added for the SCL form of the ladder/FBD networks
      _w1 : Bool;
      _w2 : Bool;
      _w3 : Bool;
      _w4 : Bool;
      _w5 : Bool;
      _w6 : Bool;
      _w7 : Bool;
      _w8 : Bool;
   END_VAR
BEGIN

REGION Network 1
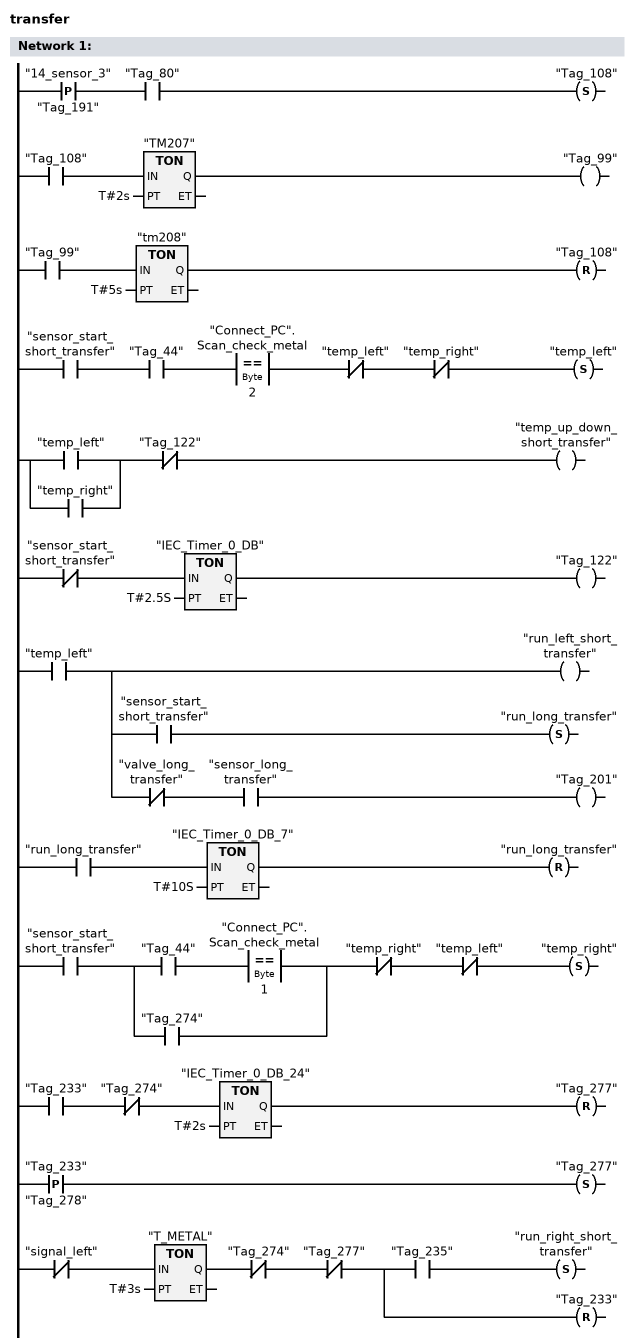
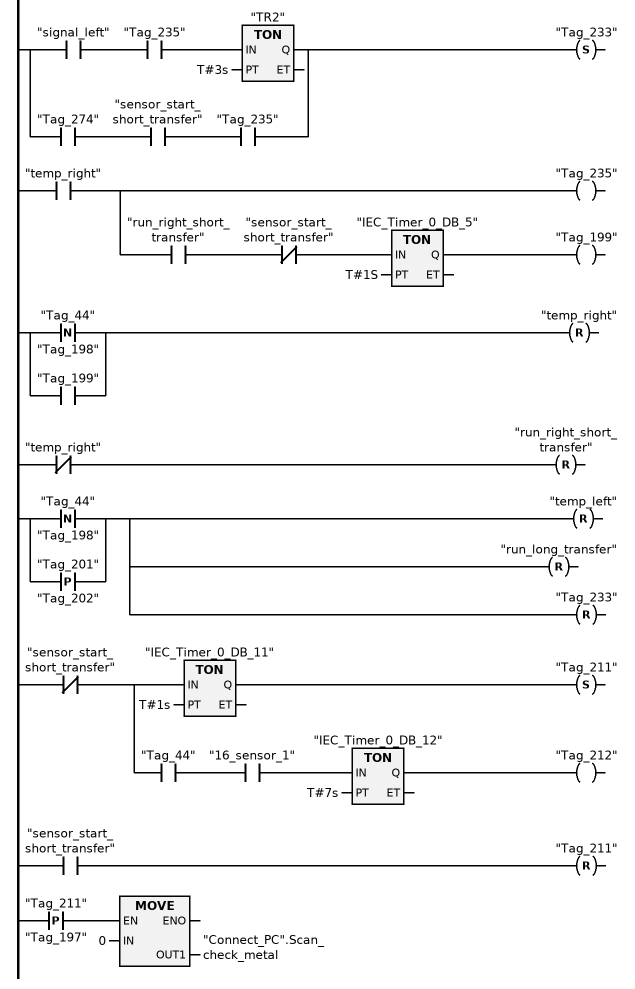
   #_w1 := "14_sensor_3" AND NOT "Tag_191";   // rising edge of "14_sensor_3"
   "Tag_191" := "14_sensor_3";
   IF #_w1 AND "Tag_80" THEN "Tag_108" := TRUE; END_IF;
   "TM207".TON(IN := "Tag_108", PT := T#2s);
   "Tag_99" := "TM207".Q;
   "tm208".TON(IN := "Tag_99", PT := T#5s);
   IF "tm208".Q THEN "Tag_108" := FALSE; END_IF;
   IF "sensor_start_short_transfer" AND "Tag_44" AND ("Connect_PC".Scan_check_metal = 2) AND NOT "temp_left" AND NOT "temp_right" THEN
       "temp_left" := TRUE;
   END_IF;
   "temp_up_down_short_transfer" := ("temp_left" OR "temp_right") AND NOT "Tag_122";
   "IEC_Timer_0_DB".TON(IN := NOT "sensor_start_short_transfer", PT := T#2.5S);
   "Tag_122" := "IEC_Timer_0_DB".Q;
   "run_left_short_transfer" := "temp_left";
   IF "temp_left" AND "sensor_start_short_transfer" THEN "run_long_transfer" := TRUE; END_IF;
   "Tag_201" := "temp_left" AND NOT "valve_long_transfer" AND "sensor_long_transfer";
   "IEC_Timer_0_DB_7".TON(IN := "run_long_transfer", PT := T#10S);
   IF "IEC_Timer_0_DB_7".Q THEN "run_long_transfer" := FALSE; END_IF;
   IF "sensor_start_short_transfer" AND (("Tag_44" AND ("Connect_PC".Scan_check_metal = 1)) OR "Tag_274") AND NOT "temp_right" AND NOT "temp_left" THEN
       "temp_right" := TRUE;
   END_IF;
   "IEC_Timer_0_DB_24".TON(IN := "Tag_233" AND NOT "Tag_274", PT := T#2s);
   IF "IEC_Timer_0_DB_24".Q THEN "Tag_277" := FALSE; END_IF;
   #_w2 := "Tag_233" AND NOT "Tag_278";   // rising edge of "Tag_233"
   "Tag_278" := "Tag_233";
   IF #_w2 THEN "Tag_277" := TRUE; END_IF;
   "T_METAL".TON(IN := NOT "signal_left", PT := T#3s);
   #_w3 := "T_METAL".Q AND NOT "Tag_274" AND NOT "Tag_277";
   IF #_w3 AND "Tag_235" THEN "run_right_short_transfer" := TRUE; END_IF;
   IF #_w3 THEN "Tag_233" := FALSE; END_IF;
   "TR2".TON(IN := "signal_left" AND "Tag_235", PT := T#3s);
   IF "TR2".Q OR ("Tag_274" AND "sensor_start_short_transfer" AND "Tag_235") THEN "Tag_233" := TRUE; END_IF;
   "Tag_235" := "temp_right";
   "IEC_Timer_0_DB_5".TON(IN := "temp_right" AND "run_right_short_transfer" AND NOT "sensor_start_short_transfer",
                          PT := T#1S);
   "Tag_199" := "IEC_Timer_0_DB_5".Q;
   #_w4 := NOT "Tag_44" AND "Tag_198";   // falling edge of "Tag_44"
   "Tag_198" := "Tag_44";
   IF #_w4 OR "Tag_199" THEN "temp_right" := FALSE; END_IF;
   IF NOT "temp_right" THEN "run_right_short_transfer" := FALSE; END_IF;
   #_w5 := NOT "Tag_44" AND "Tag_198";   // falling edge of "Tag_44"
   "Tag_198" := "Tag_44";
   #_w6 := "Tag_201" AND NOT "Tag_202";   // rising edge of "Tag_201"
   "Tag_202" := "Tag_201";
   IF #_w5 OR #_w6 THEN
       "temp_left" := FALSE;
       "run_long_transfer" := FALSE;
       "Tag_233" := FALSE;
   END_IF;
   #_w7 := NOT "sensor_start_short_transfer";
   "IEC_Timer_0_DB_11".TON(IN := #_w7, PT := T#1s);
   IF "IEC_Timer_0_DB_11".Q THEN "Tag_211" := TRUE; END_IF;
   "IEC_Timer_0_DB_12".TON(IN := #_w7 AND "Tag_44" AND "16_sensor_1", PT := T#7s);
   "Tag_212" := "IEC_Timer_0_DB_12".Q;
   IF "sensor_start_short_transfer" THEN "Tag_211" := FALSE; END_IF;
   #_w8 := "Tag_211" AND NOT "Tag_197";   // rising edge of "Tag_211"
   "Tag_197" := "Tag_211";
   IF #_w8 THEN "Connect_PC".Scan_check_metal := 0; END_IF;
END_REGION
END_FUNCTION

FUNCTION "pusher" : Void   // FC2, LAD
{ S7_Optimized_Access := 'TRUE' }
VERSION : 0.1
   VAR_TEMP   // added for the SCL form of the ladder/FBD networks
      _w1 : Bool;
      _w2 : Bool;
      _w3 : Bool;
      _w4 : Bool;
      _w5 : Bool;
      _w6 : Bool;
      _w7 : Bool;
      _w8 : Bool;
   END_VAR
BEGIN

REGION Network 1
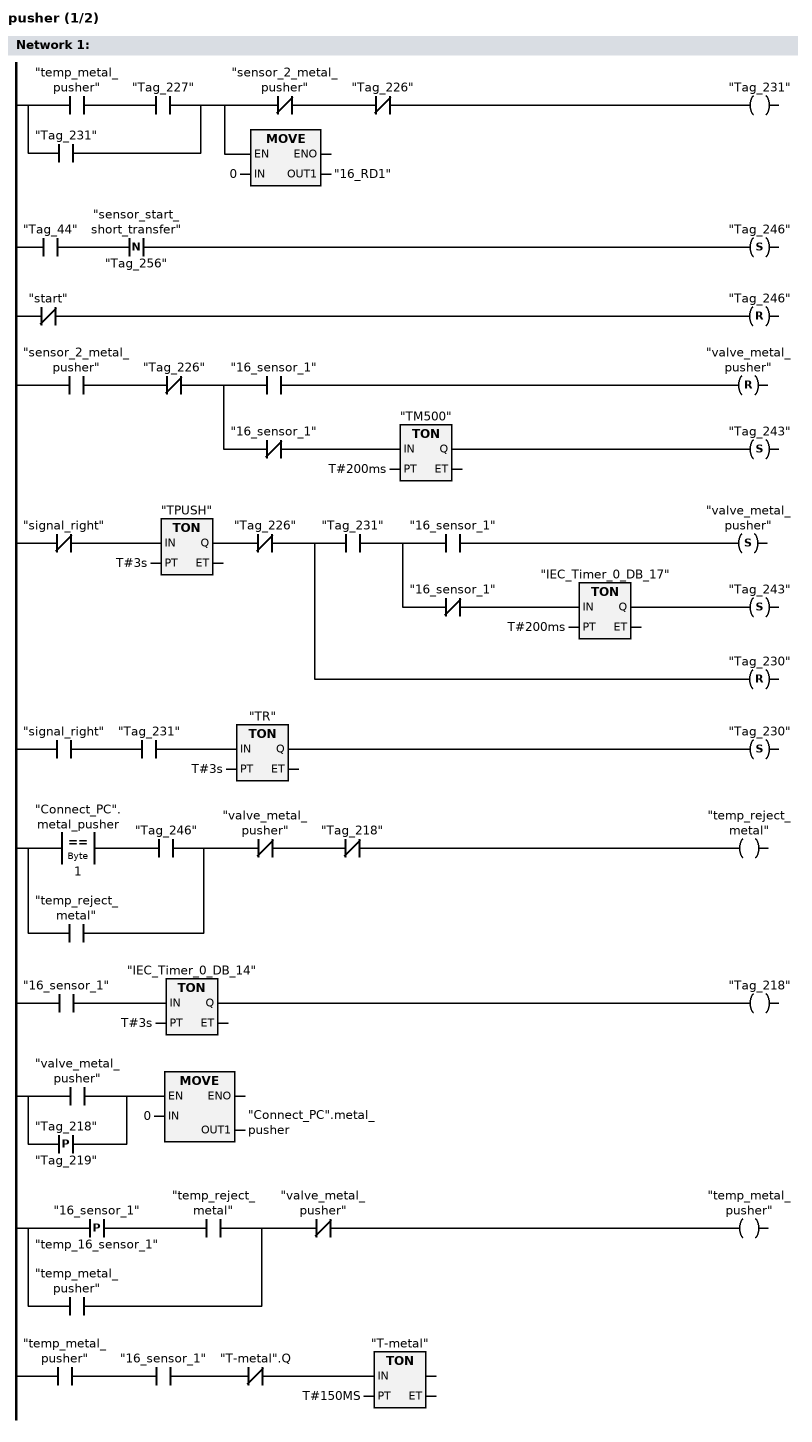
   #_w1 := ("temp_metal_pusher" AND "Tag_227") OR "Tag_231";
   "Tag_231" := #_w1 AND NOT "sensor_2_metal_pusher" AND NOT "Tag_226";
   IF #_w1 THEN "16_RD1" := 0; END_IF;
   #_w2 := "Tag_44" AND NOT "sensor_start_short_transfer" AND "Tag_256";   // falling edge of "sensor_start_short_transfer"
   "Tag_256" := "sensor_start_short_transfer";
   IF #_w2 THEN "Tag_246" := TRUE; END_IF;
   IF NOT "start" THEN "Tag_246" := FALSE; END_IF;
   #_w3 := "sensor_2_metal_pusher" AND NOT "Tag_226";
   IF #_w3 AND "16_sensor_1" THEN "valve_metal_pusher" := FALSE; END_IF;
   "TM500".TON(IN := #_w3 AND NOT "16_sensor_1", PT := T#200ms);
   IF "TM500".Q THEN "Tag_243" := TRUE; END_IF;
   "TPUSH".TON(IN := NOT "signal_right", PT := T#3s);
   #_w4 := "TPUSH".Q AND NOT "Tag_226";
   #_w5 := #_w4 AND "Tag_231";
   IF #_w5 AND "16_sensor_1" THEN "valve_metal_pusher" := TRUE; END_IF;
   "IEC_Timer_0_DB_17".TON(IN := #_w5 AND NOT "16_sensor_1", PT := T#200ms);
   IF "IEC_Timer_0_DB_17".Q THEN "Tag_243" := TRUE; END_IF;
   IF #_w4 THEN "Tag_230" := FALSE; END_IF;
   "TR".TON(IN := "signal_right" AND "Tag_231", PT := T#3s);
   IF "TR".Q THEN "Tag_230" := TRUE; END_IF;
   "temp_reject_metal" := ((("Connect_PC".metal_pusher = 1) AND "Tag_246") OR "temp_reject_metal") AND NOT "valve_metal_pusher" AND NOT "Tag_218";
   "IEC_Timer_0_DB_14".TON(IN := "16_sensor_1", PT := T#3s);
   "Tag_218" := "IEC_Timer_0_DB_14".Q;
   #_w6 := "Tag_218" AND NOT "Tag_219";   // rising edge of "Tag_218"
   "Tag_219" := "Tag_218";
   IF "valve_metal_pusher" OR #_w6 THEN "Connect_PC".metal_pusher := 0; END_IF;
   #_w7 := "16_sensor_1" AND NOT "temp_16_sensor_1";   // rising edge of "16_sensor_1"
   "temp_16_sensor_1" := "16_sensor_1";
   "temp_metal_pusher" := ((#_w7 AND "temp_reject_metal") OR "temp_metal_pusher") AND NOT "valve_metal_pusher";
   "T-metal".TON(IN := "temp_metal_pusher" AND "16_sensor_1" AND NOT "T-metal".Q, PT := T#150MS);
END_REGION

REGION Network 2
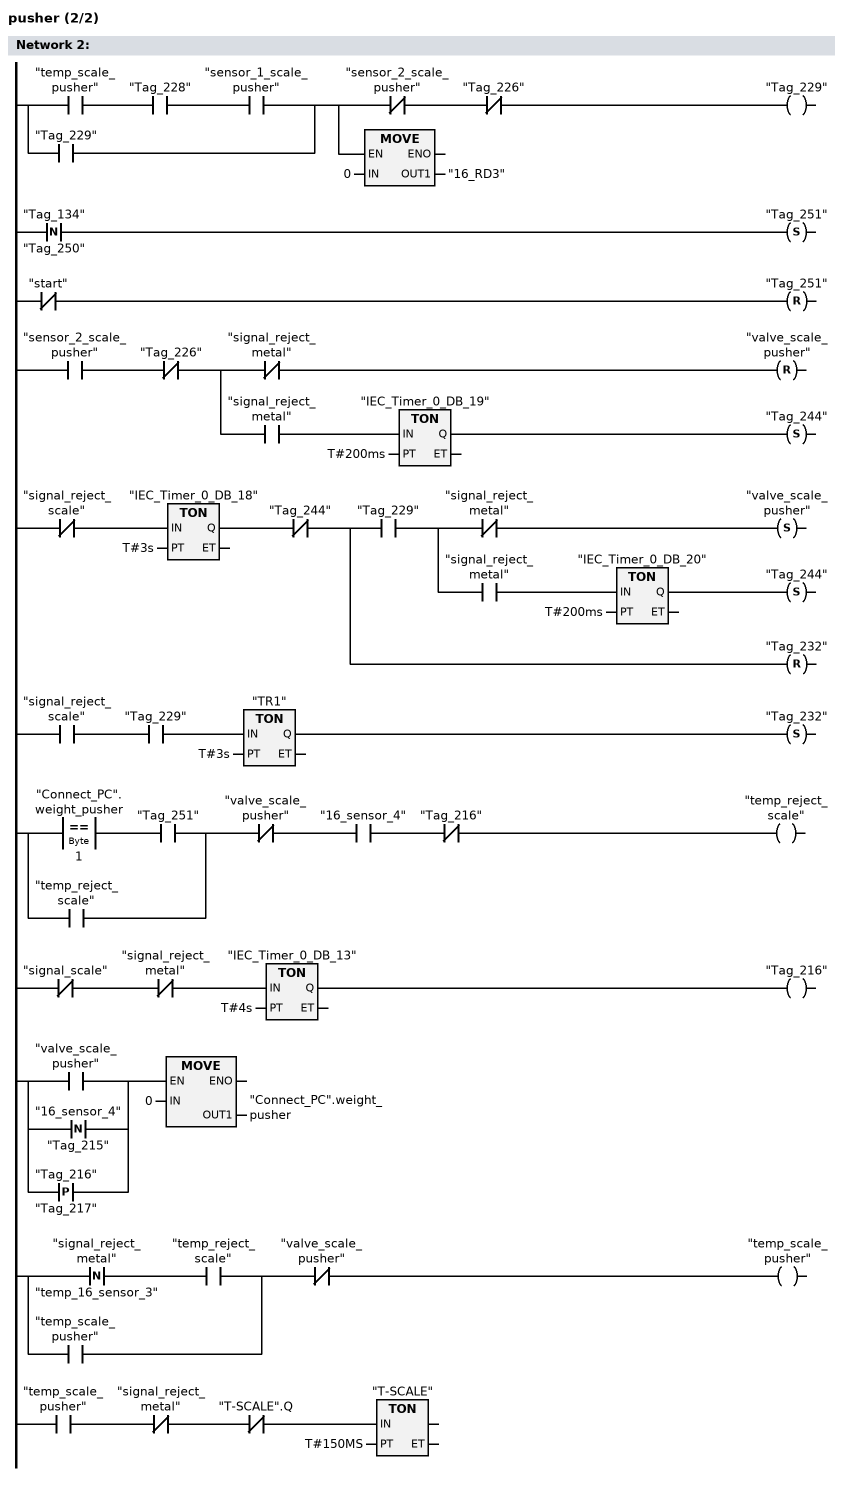
   #_w1 := ("temp_scale_pusher" AND "Tag_228" AND "sensor_1_scale_pusher") OR "Tag_229";
   "Tag_229" := #_w1 AND NOT "sensor_2_scale_pusher" AND NOT "Tag_226";
   IF #_w1 THEN "16_RD3" := 0; END_IF;
   #_w2 := NOT "Tag_134" AND "Tag_250";   // falling edge of "Tag_134"
   "Tag_250" := "Tag_134";
   IF #_w2 THEN "Tag_251" := TRUE; END_IF;
   IF NOT "start" THEN "Tag_251" := FALSE; END_IF;
   #_w3 := "sensor_2_scale_pusher" AND NOT "Tag_226";
   IF #_w3 AND NOT "signal_reject_metal" THEN "valve_scale_pusher" := FALSE; END_IF;
   "IEC_Timer_0_DB_19".TON(IN := #_w3 AND "signal_reject_metal", PT := T#200ms);
   IF "IEC_Timer_0_DB_19".Q THEN "Tag_244" := TRUE; END_IF;
   "IEC_Timer_0_DB_18".TON(IN := NOT "signal_reject_scale", PT := T#3s);
   #_w4 := "IEC_Timer_0_DB_18".Q AND NOT "Tag_244";
   #_w5 := #_w4 AND "Tag_229";
   IF #_w5 AND NOT "signal_reject_metal" THEN "valve_scale_pusher" := TRUE; END_IF;
   "IEC_Timer_0_DB_20".TON(IN := #_w5 AND "signal_reject_metal", PT := T#200ms);
   IF "IEC_Timer_0_DB_20".Q THEN "Tag_244" := TRUE; END_IF;
   IF #_w4 THEN "Tag_232" := FALSE; END_IF;
   "TR1".TON(IN := "signal_reject_scale" AND "Tag_229", PT := T#3s);
   IF "TR1".Q THEN "Tag_232" := TRUE; END_IF;
   "temp_reject_scale" := ((("Connect_PC".weight_pusher = 1) AND "Tag_251") OR "temp_reject_scale") AND NOT "valve_scale_pusher" AND "16_sensor_4" AND NOT "Tag_216";
   "IEC_Timer_0_DB_13".TON(IN := NOT "signal_scale" AND NOT "signal_reject_metal", PT := T#4s);
   "Tag_216" := "IEC_Timer_0_DB_13".Q;
   #_w6 := NOT "16_sensor_4" AND "Tag_215";   // falling edge of "16_sensor_4"
   "Tag_215" := "16_sensor_4";
   #_w7 := "Tag_216" AND NOT "Tag_217";   // rising edge of "Tag_216"
   "Tag_217" := "Tag_216";
   IF "valve_scale_pusher" OR #_w6 OR #_w7 THEN "Connect_PC".weight_pusher := 0; END_IF;
   #_w8 := NOT "signal_reject_metal" AND "temp_16_sensor_3";   // falling edge of "signal_reject_metal"
   "temp_16_sensor_3" := "signal_reject_metal";
   "temp_scale_pusher" := ((#_w8 AND "temp_reject_scale") OR "temp_scale_pusher") AND NOT "valve_scale_pusher";
   "T-SCALE".TON(IN := "temp_scale_pusher" AND NOT "signal_reject_metal" AND NOT "T-SCALE".Q, PT := T#150MS);
END_REGION
END_FUNCTION

FUNCTION "192.168.80.13" : Void   // FC3, LAD
{ S7_Optimized_Access := 'TRUE' }
VERSION : 0.1
   VAR_TEMP   // added for the SCL form of the ladder/FBD networks
      _w1 : Bool;
      _w2 : Bool;
      _w3 : Bool;
      _w4 : Bool;
   END_VAR
BEGIN

REGION Network 1: Zone 4
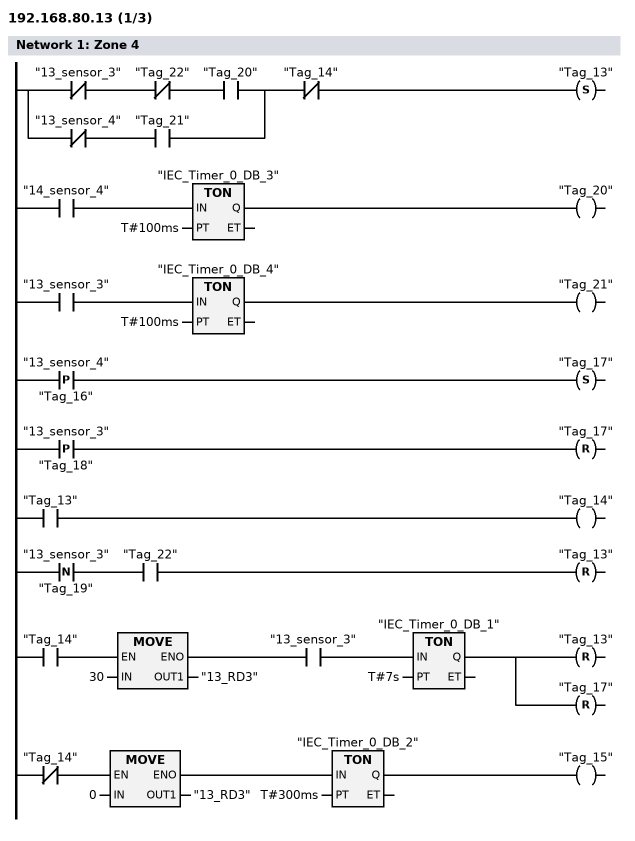
   IF ((NOT "13_sensor_3" AND NOT "Tag_22" AND "Tag_20") OR (NOT "13_sensor_4" AND "Tag_21")) AND NOT "Tag_14" THEN
       "Tag_13" := TRUE;
   END_IF;
   "IEC_Timer_0_DB_3".TON(IN := "14_sensor_4", PT := T#100ms);
   "Tag_20" := "IEC_Timer_0_DB_3".Q;
   "IEC_Timer_0_DB_4".TON(IN := "13_sensor_3", PT := T#100ms);
   "Tag_21" := "IEC_Timer_0_DB_4".Q;
   #_w1 := "13_sensor_4" AND NOT "Tag_16";   // rising edge of "13_sensor_4"
   "Tag_16" := "13_sensor_4";
   IF #_w1 THEN "Tag_17" := TRUE; END_IF;
   #_w2 := "13_sensor_3" AND NOT "Tag_18";   // rising edge of "13_sensor_3"
   "Tag_18" := "13_sensor_3";
   IF #_w2 THEN "Tag_17" := FALSE; END_IF;
   "Tag_14" := "Tag_13";
   #_w3 := NOT "13_sensor_3" AND "Tag_19";   // falling edge of "13_sensor_3"
   "Tag_19" := "13_sensor_3";
   IF #_w3 AND "Tag_22" THEN "Tag_13" := FALSE; END_IF;
   IF "Tag_14" THEN "13_RD3" := 30; END_IF;
   "IEC_Timer_0_DB_1".TON(IN := "Tag_14" AND "13_sensor_3", PT := T#7s);
   IF "IEC_Timer_0_DB_1".Q THEN
       "Tag_13" := FALSE;
       "Tag_17" := FALSE;
   END_IF;
   IF NOT "Tag_14" THEN "13_RD3" := 0; END_IF;
   "IEC_Timer_0_DB_2".TON(IN := NOT "Tag_14", PT := T#300ms);
   "Tag_15" := "IEC_Timer_0_DB_2".Q;
END_REGION

REGION Network 2: Zone 3
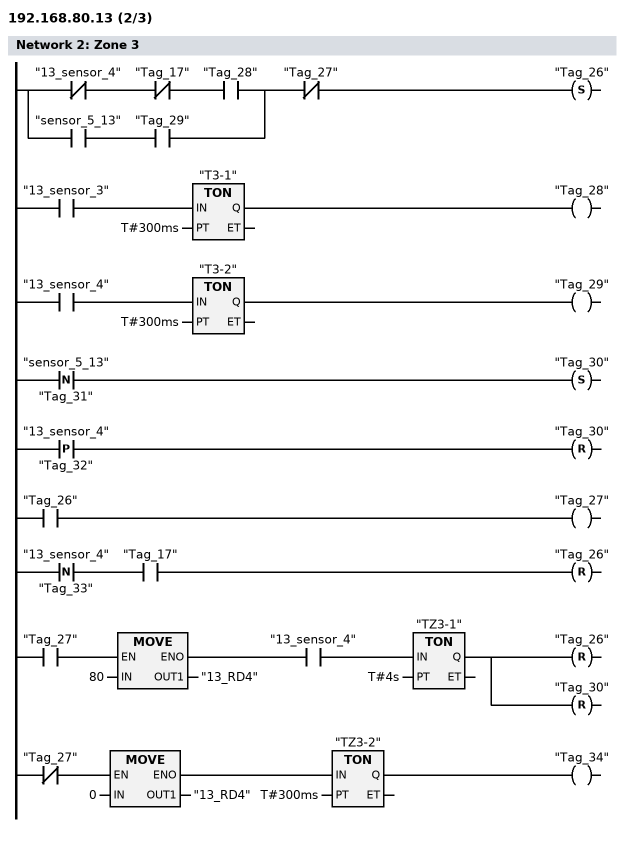
   IF ((NOT "13_sensor_4" AND NOT "Tag_17" AND "Tag_28") OR ("sensor_5_13" AND "Tag_29")) AND NOT "Tag_27" THEN
       "Tag_26" := TRUE;
   END_IF;
   "T3-1".TON(IN := "13_sensor_3", PT := T#300ms);
   "Tag_28" := "T3-1".Q;
   "T3-2".TON(IN := "13_sensor_4", PT := T#300ms);
   "Tag_29" := "T3-2".Q;
   #_w1 := NOT "sensor_5_13" AND "Tag_31";   // falling edge of "sensor_5_13"
   "Tag_31" := "sensor_5_13";
   IF #_w1 THEN "Tag_30" := TRUE; END_IF;
   #_w2 := "13_sensor_4" AND NOT "Tag_32";   // rising edge of "13_sensor_4"
   "Tag_32" := "13_sensor_4";
   IF #_w2 THEN "Tag_30" := FALSE; END_IF;
   "Tag_27" := "Tag_26";
   #_w3 := NOT "13_sensor_4" AND "Tag_33";   // falling edge of "13_sensor_4"
   "Tag_33" := "13_sensor_4";
   IF #_w3 AND "Tag_17" THEN "Tag_26" := FALSE; END_IF;
   IF "Tag_27" THEN "13_RD4" := 80; END_IF;
   "TZ3-1".TON(IN := "Tag_27" AND "13_sensor_4", PT := T#4s);
   IF "TZ3-1".Q THEN
       "Tag_26" := FALSE;
       "Tag_30" := FALSE;
   END_IF;
   IF NOT "Tag_27" THEN "13_RD4" := 0; END_IF;
   "TZ3-2".TON(IN := NOT "Tag_27", PT := T#300ms);
   "Tag_34" := "TZ3-2".Q;
END_REGION

REGION Network 3: Zone 2
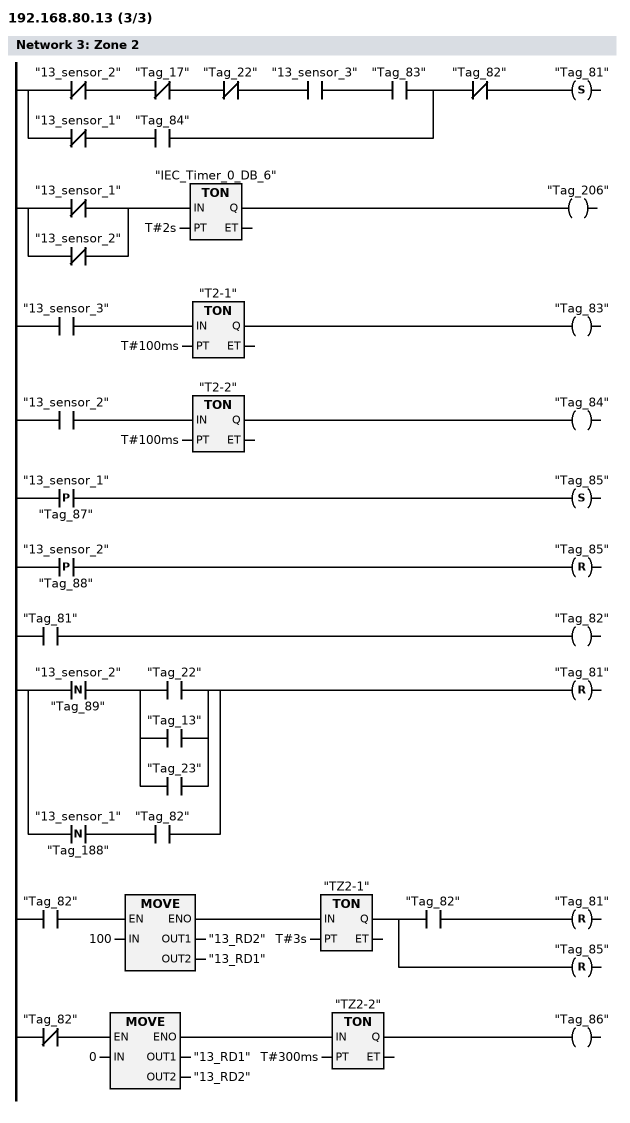
   IF ((NOT "13_sensor_2" AND NOT "Tag_17" AND NOT "Tag_22" AND "13_sensor_3" AND "Tag_83") OR (NOT "13_sensor_1" AND "Tag_84")) AND NOT "Tag_82" THEN
       "Tag_81" := TRUE;
   END_IF;
   "IEC_Timer_0_DB_6".TON(IN := NOT "13_sensor_1" OR NOT "13_sensor_2", PT := T#2s);
   "Tag_206" := "IEC_Timer_0_DB_6".Q;
   "T2-1".TON(IN := "13_sensor_3", PT := T#100ms);
   "Tag_83" := "T2-1".Q;
   "T2-2".TON(IN := "13_sensor_2", PT := T#100ms);
   "Tag_84" := "T2-2".Q;
   #_w1 := "13_sensor_1" AND NOT "Tag_87";   // rising edge of "13_sensor_1"
   "Tag_87" := "13_sensor_1";
   IF #_w1 THEN "Tag_85" := TRUE; END_IF;
   #_w2 := "13_sensor_2" AND NOT "Tag_88";   // rising edge of "13_sensor_2"
   "Tag_88" := "13_sensor_2";
   IF #_w2 THEN "Tag_85" := FALSE; END_IF;
   "Tag_82" := "Tag_81";
   #_w3 := NOT "13_sensor_2" AND "Tag_89";   // falling edge of "13_sensor_2"
   "Tag_89" := "13_sensor_2";
   #_w4 := NOT "13_sensor_1" AND "Tag_188";   // falling edge of "13_sensor_1"
   "Tag_188" := "13_sensor_1";
   IF (#_w3 AND ("Tag_22" OR "Tag_13" OR "Tag_23")) OR (#_w4 AND "Tag_82") THEN "Tag_81" := FALSE; END_IF;
   IF "Tag_82" THEN
       "13_RD2" := 100;
       "13_RD1" := 100;
   END_IF;
   "TZ2-1".TON(IN := "Tag_82", PT := T#3s);
   IF "TZ2-1".Q AND "Tag_82" THEN "Tag_81" := FALSE; END_IF;
   IF "TZ2-1".Q THEN "Tag_85" := FALSE; END_IF;
   IF NOT "Tag_82" THEN
       "13_RD1" := 0;
       "13_RD2" := 0;
   END_IF;
   "TZ2-2".TON(IN := NOT "Tag_82", PT := T#300ms);
   "Tag_86" := "TZ2-2".Q;
END_REGION
END_FUNCTION

FUNCTION "192.168.80.14" : Void   // FC4, LAD
{ S7_Optimized_Access := 'TRUE' }
VERSION : 0.1
   VAR_TEMP   // added for the SCL form of the ladder/FBD networks
      _w1 : Bool;
      _w2 : Bool;
      _w3 : Bool;
      _w4 : Bool;
      _w5 : Bool;
      _w6 : Bool;
      _w7 : Bool;
      _w8 : Bool;
      _w9 : Bool;
   END_VAR
BEGIN

REGION Network 1: Zone 5
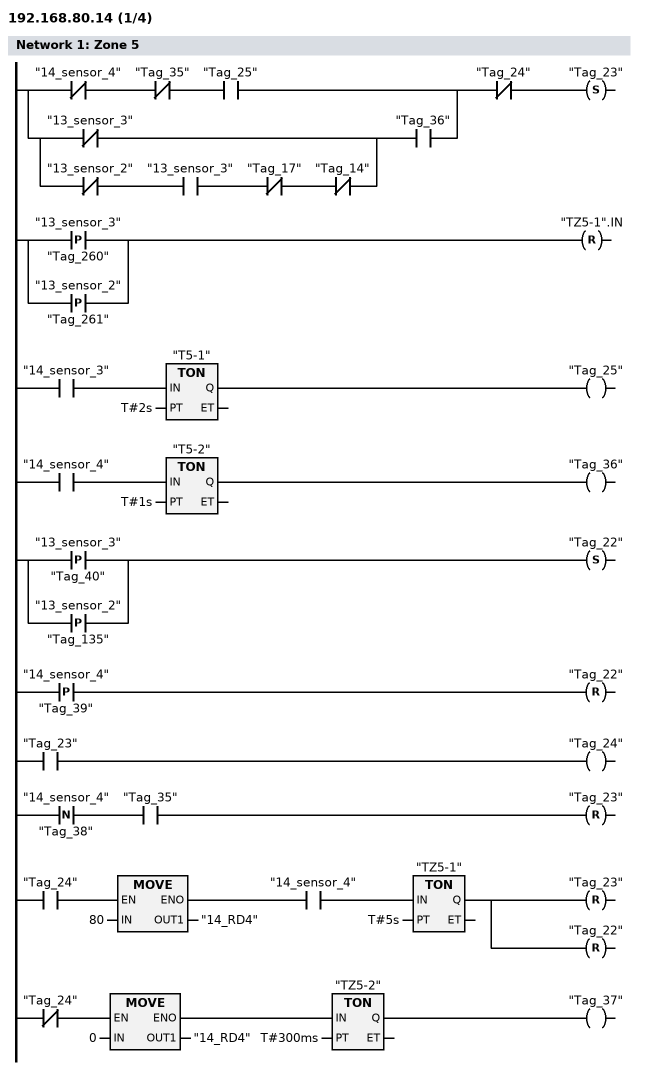
   IF ((NOT "14_sensor_4" AND NOT "Tag_35" AND "Tag_25") OR ((NOT "13_sensor_3" OR (NOT "13_sensor_2" AND "13_sensor_3" AND NOT "Tag_17" AND NOT "Tag_14")) AND "Tag_36")) AND NOT "Tag_24" THEN
       "Tag_23" := TRUE;
   END_IF;
   #_w1 := "13_sensor_3" AND NOT "Tag_260";   // rising edge of "13_sensor_3"
   "Tag_260" := "13_sensor_3";
   #_w2 := "13_sensor_2" AND NOT "Tag_261";   // rising edge of "13_sensor_2"
   "Tag_261" := "13_sensor_2";
   IF #_w1 OR #_w2 THEN "TZ5-1".IN := FALSE; END_IF;
   "T5-1".TON(IN := "14_sensor_3", PT := T#2s);
   "Tag_25" := "T5-1".Q;
   "T5-2".TON(IN := "14_sensor_4", PT := T#1s);
   "Tag_36" := "T5-2".Q;
   #_w3 := "13_sensor_3" AND NOT "Tag_40";   // rising edge of "13_sensor_3"
   "Tag_40" := "13_sensor_3";
   #_w4 := "13_sensor_2" AND NOT "Tag_135";   // rising edge of "13_sensor_2"
   "Tag_135" := "13_sensor_2";
   IF #_w3 OR #_w4 THEN "Tag_22" := TRUE; END_IF;
   #_w5 := "14_sensor_4" AND NOT "Tag_39";   // rising edge of "14_sensor_4"
   "Tag_39" := "14_sensor_4";
   IF #_w5 THEN "Tag_22" := FALSE; END_IF;
   "Tag_24" := "Tag_23";
   #_w6 := NOT "14_sensor_4" AND "Tag_38";   // falling edge of "14_sensor_4"
   "Tag_38" := "14_sensor_4";
   IF #_w6 AND "Tag_35" THEN "Tag_23" := FALSE; END_IF;
   IF "Tag_24" THEN "14_RD4" := 80; END_IF;
   "TZ5-1".TON(IN := "Tag_24" AND "14_sensor_4", PT := T#5s);
   IF "TZ5-1".Q THEN
       "Tag_23" := FALSE;
       "Tag_22" := FALSE;
   END_IF;
   IF NOT "Tag_24" THEN "14_RD4" := 0; END_IF;
   "TZ5-2".TON(IN := NOT "Tag_24", PT := T#300ms);
   "Tag_37" := "TZ5-2".Q;
END_REGION

REGION Network 2: Zone 6
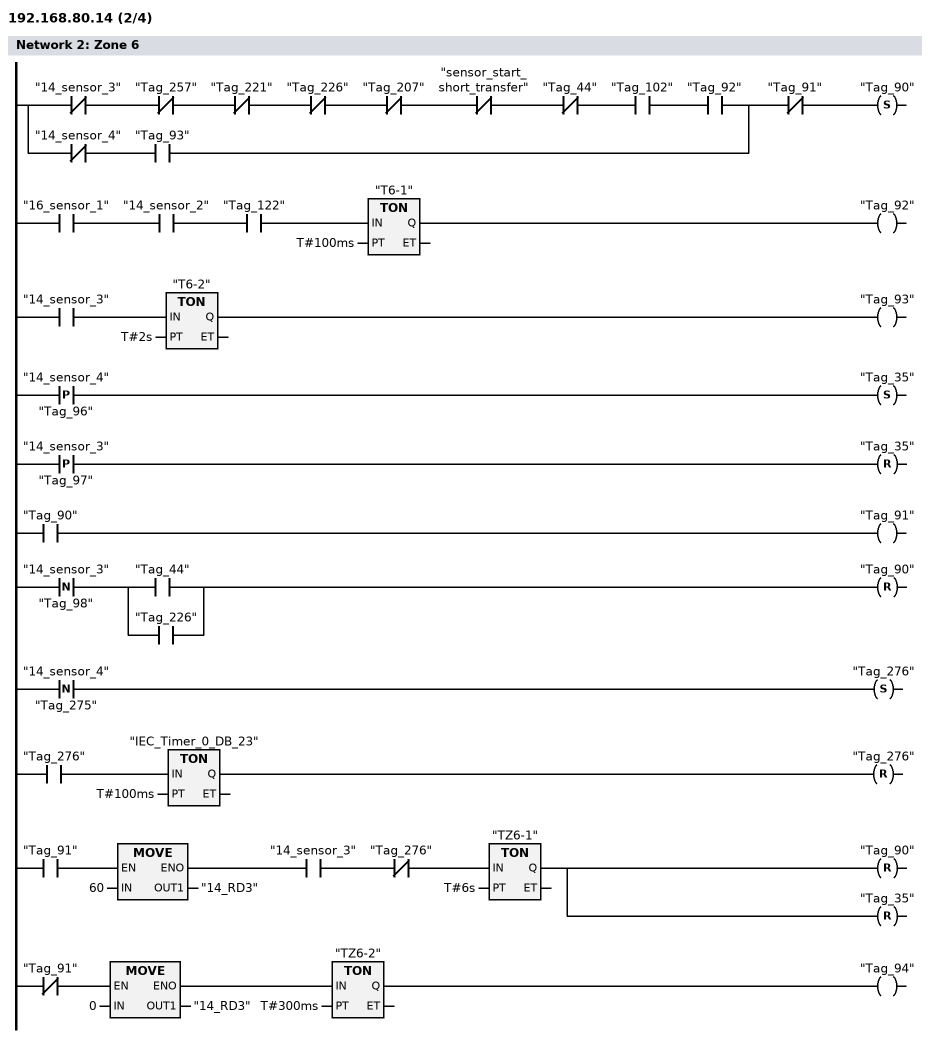
   IF ((NOT "14_sensor_3" AND NOT "Tag_257" AND NOT "Tag_221" AND NOT "Tag_226" AND NOT "Tag_207" AND NOT "sensor_start_short_transfer" AND NOT "Tag_44" AND "Tag_102" AND "Tag_92") OR (NOT "14_sensor_4" AND "Tag_93")) AND NOT "Tag_91" THEN
       "Tag_90" := TRUE;
   END_IF;
   "T6-1".TON(IN := "16_sensor_1" AND "14_sensor_2" AND "Tag_122", PT := T#100ms);
   "Tag_92" := "T6-1".Q;
   "T6-2".TON(IN := "14_sensor_3", PT := T#2s);
   "Tag_93" := "T6-2".Q;
   #_w1 := "14_sensor_4" AND NOT "Tag_96";   // rising edge of "14_sensor_4"
   "Tag_96" := "14_sensor_4";
   IF #_w1 THEN "Tag_35" := TRUE; END_IF;
   #_w2 := "14_sensor_3" AND NOT "Tag_97";   // rising edge of "14_sensor_3"
   "Tag_97" := "14_sensor_3";
   IF #_w2 THEN "Tag_35" := FALSE; END_IF;
   "Tag_91" := "Tag_90";
   #_w3 := NOT "14_sensor_3" AND "Tag_98";   // falling edge of "14_sensor_3"
   "Tag_98" := "14_sensor_3";
   IF #_w3 AND ("Tag_44" OR "Tag_226") THEN "Tag_90" := FALSE; END_IF;
   #_w4 := NOT "14_sensor_4" AND "Tag_275";   // falling edge of "14_sensor_4"
   "Tag_275" := "14_sensor_4";
   IF #_w4 THEN "Tag_276" := TRUE; END_IF;
   "IEC_Timer_0_DB_23".TON(IN := "Tag_276", PT := T#100ms);
   IF "IEC_Timer_0_DB_23".Q THEN "Tag_276" := FALSE; END_IF;
   IF "Tag_91" THEN "14_RD3" := 60; END_IF;
   "TZ6-1".TON(IN := "Tag_91" AND "14_sensor_3" AND NOT "Tag_276", PT := T#6s);
   IF "TZ6-1".Q THEN
       "Tag_90" := FALSE;
       "Tag_35" := FALSE;
   END_IF;
   IF NOT "Tag_91" THEN "14_RD3" := 0; END_IF;
   "TZ6-2".TON(IN := NOT "Tag_91", PT := T#300ms);
   "Tag_94" := "TZ6-2".Q;
END_REGION

REGION Network 3: Zone 7
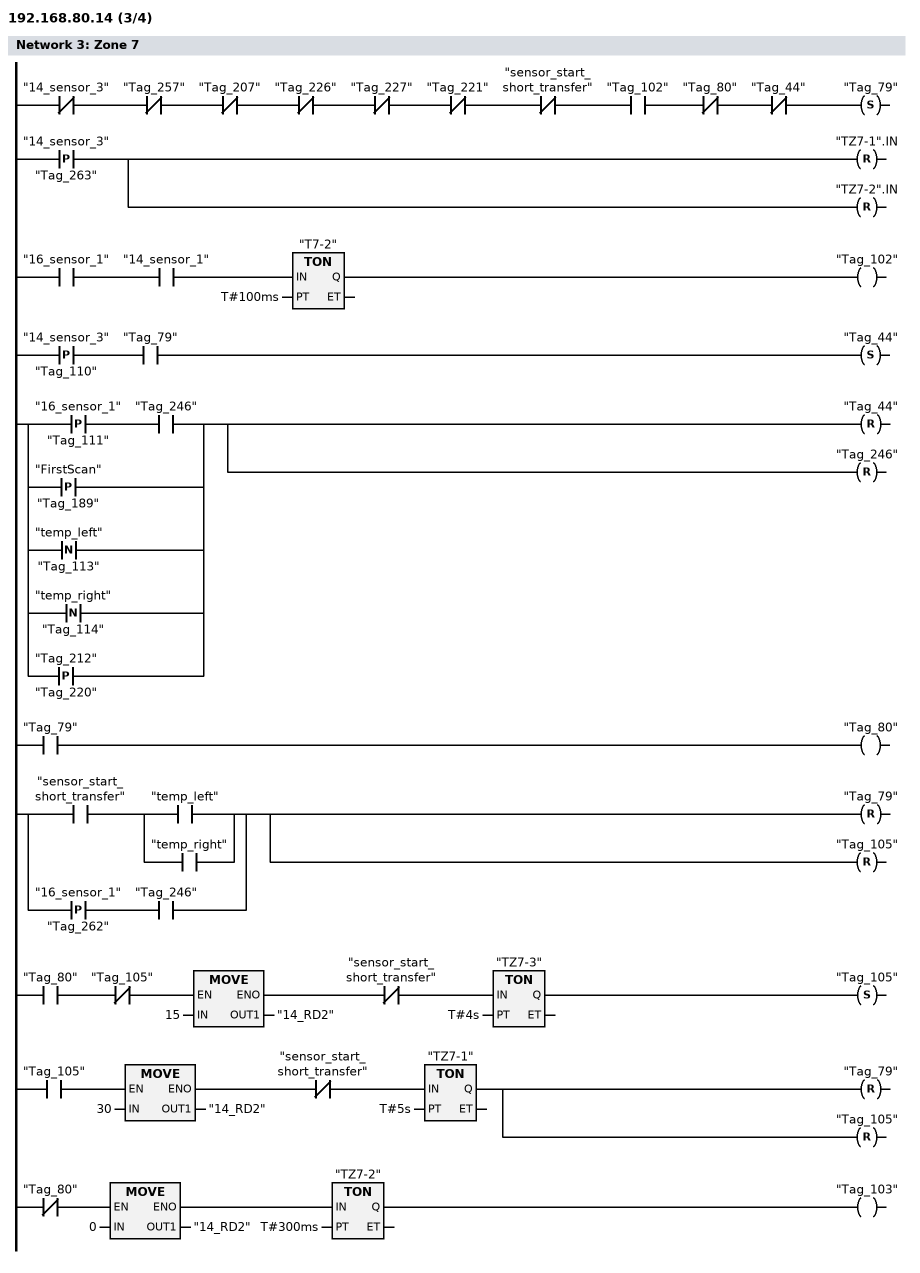
   IF NOT "14_sensor_3" AND NOT "Tag_257" AND NOT "Tag_207" AND NOT "Tag_226" AND NOT "Tag_227" AND NOT "Tag_221" AND NOT "sensor_start_short_transfer" AND "Tag_102" AND NOT "Tag_80" AND NOT "Tag_44" THEN
       "Tag_79" := TRUE;
   END_IF;
   #_w1 := "14_sensor_3" AND NOT "Tag_263";   // rising edge of "14_sensor_3"
   "Tag_263" := "14_sensor_3";
   IF #_w1 THEN
       "TZ7-1".IN := FALSE;
       "TZ7-2".IN := FALSE;
   END_IF;
   "T7-2".TON(IN := "16_sensor_1" AND "14_sensor_1", PT := T#100ms);
   "Tag_102" := "T7-2".Q;
   #_w2 := "14_sensor_3" AND NOT "Tag_110";   // rising edge of "14_sensor_3"
   "Tag_110" := "14_sensor_3";
   IF #_w2 AND "Tag_79" THEN "Tag_44" := TRUE; END_IF;
   #_w3 := "16_sensor_1" AND NOT "Tag_111";   // rising edge of "16_sensor_1"
   "Tag_111" := "16_sensor_1";
   #_w4 := "FirstScan" AND NOT "Tag_189";   // rising edge of "FirstScan"
   "Tag_189" := "FirstScan";
   #_w5 := NOT "temp_left" AND "Tag_113";   // falling edge of "temp_left"
   "Tag_113" := "temp_left";
   #_w6 := NOT "temp_right" AND "Tag_114";   // falling edge of "temp_right"
   "Tag_114" := "temp_right";
   #_w7 := "Tag_212" AND NOT "Tag_220";   // rising edge of "Tag_212"
   "Tag_220" := "Tag_212";
   IF (#_w3 AND "Tag_246") OR #_w4 OR #_w5 OR #_w6 OR #_w7 THEN
       "Tag_44" := FALSE;
       "Tag_246" := FALSE;
   END_IF;
   "Tag_80" := "Tag_79";
   #_w8 := "16_sensor_1" AND NOT "Tag_262";   // rising edge of "16_sensor_1"
   "Tag_262" := "16_sensor_1";
   IF ("sensor_start_short_transfer" AND ("temp_left" OR "temp_right")) OR (#_w8 AND "Tag_246") THEN
       "Tag_79" := FALSE;
       "Tag_105" := FALSE;
   END_IF;
   #_w9 := "Tag_80" AND NOT "Tag_105";
   IF #_w9 THEN "14_RD2" := 15; END_IF;
   "TZ7-3".TON(IN := #_w9 AND NOT "sensor_start_short_transfer", PT := T#4s);
   IF "TZ7-3".Q THEN "Tag_105" := TRUE; END_IF;
   IF "Tag_105" THEN "14_RD2" := 30; END_IF;
   "TZ7-1".TON(IN := "Tag_105" AND NOT "sensor_start_short_transfer", PT := T#5s);
   IF "TZ7-1".Q THEN
       "Tag_79" := FALSE;
       "Tag_105" := FALSE;
   END_IF;
   IF NOT "Tag_80" THEN "14_RD2" := 0; END_IF;
   "TZ7-2".TON(IN := NOT "Tag_80", PT := T#300ms);
   "Tag_103" := "TZ7-2".Q;
END_REGION

REGION Network 4: Zone 8
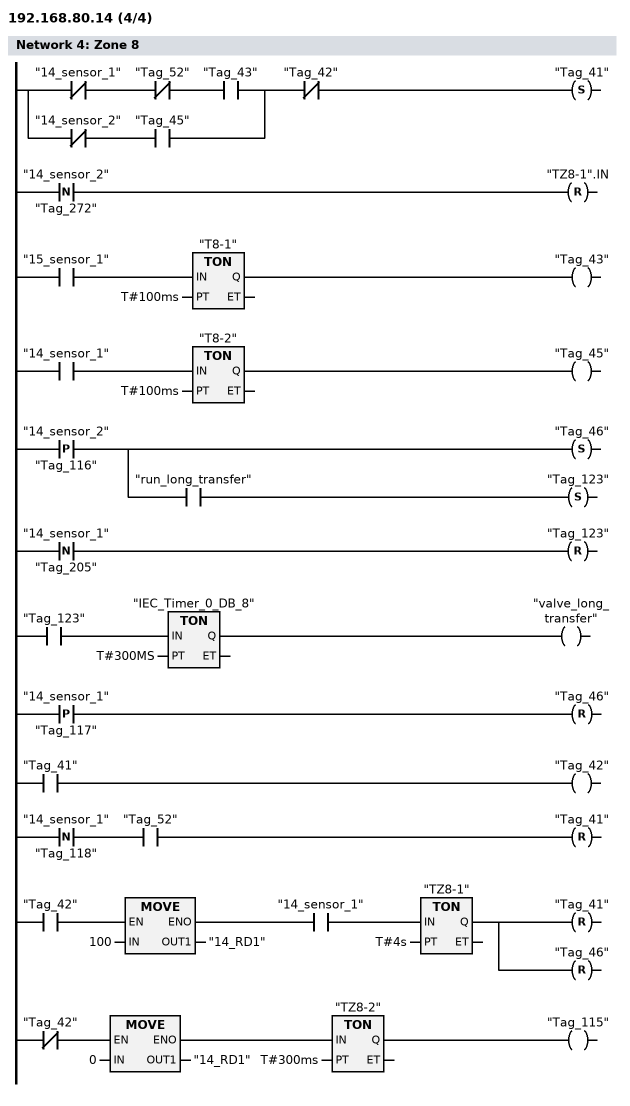
   IF ((NOT "14_sensor_1" AND NOT "Tag_52" AND "Tag_43") OR (NOT "14_sensor_2" AND "Tag_45")) AND NOT "Tag_42" THEN
       "Tag_41" := TRUE;
   END_IF;
   #_w1 := NOT "14_sensor_2" AND "Tag_272";   // falling edge of "14_sensor_2"
   "Tag_272" := "14_sensor_2";
   IF #_w1 THEN "TZ8-1".IN := FALSE; END_IF;
   "T8-1".TON(IN := "15_sensor_1", PT := T#100ms);
   "Tag_43" := "T8-1".Q;
   "T8-2".TON(IN := "14_sensor_1", PT := T#100ms);
   "Tag_45" := "T8-2".Q;
   #_w2 := "14_sensor_2" AND NOT "Tag_116";   // rising edge of "14_sensor_2"
   "Tag_116" := "14_sensor_2";
   IF #_w2 THEN "Tag_46" := TRUE; END_IF;
   IF #_w2 AND "run_long_transfer" THEN "Tag_123" := TRUE; END_IF;
   #_w3 := NOT "14_sensor_1" AND "Tag_205";   // falling edge of "14_sensor_1"
   "Tag_205" := "14_sensor_1";
   IF #_w3 THEN "Tag_123" := FALSE; END_IF;
   "IEC_Timer_0_DB_8".TON(IN := "Tag_123", PT := T#300MS);
   "valve_long_transfer" := "IEC_Timer_0_DB_8".Q;
   #_w4 := "14_sensor_1" AND NOT "Tag_117";   // rising edge of "14_sensor_1"
   "Tag_117" := "14_sensor_1";
   IF #_w4 THEN "Tag_46" := FALSE; END_IF;
   "Tag_42" := "Tag_41";
   #_w5 := NOT "14_sensor_1" AND "Tag_118";   // falling edge of "14_sensor_1"
   "Tag_118" := "14_sensor_1";
   IF #_w5 AND "Tag_52" THEN "Tag_41" := FALSE; END_IF;
   IF "Tag_42" THEN "14_RD1" := 100; END_IF;
   "TZ8-1".TON(IN := "Tag_42" AND "14_sensor_1", PT := T#4s);
   IF "TZ8-1".Q THEN
       "Tag_41" := FALSE;
       "Tag_46" := FALSE;
   END_IF;
   IF NOT "Tag_42" THEN "14_RD1" := 0; END_IF;
   "TZ8-2".TON(IN := NOT "Tag_42", PT := T#300ms);
   "Tag_115" := "TZ8-2".Q;
END_REGION
END_FUNCTION

FUNCTION "192.168.80.15" : Void   // FC5, LAD
{ S7_Optimized_Access := 'TRUE' }
VERSION : 0.1
   VAR_TEMP   // added for the SCL form of the ladder/FBD networks
      _w1 : Bool;
      _w2 : Bool;
      _w3 : Bool;
      _w4 : Bool;
      _w5 : Bool;
   END_VAR
BEGIN

REGION Network 1: Zone 9
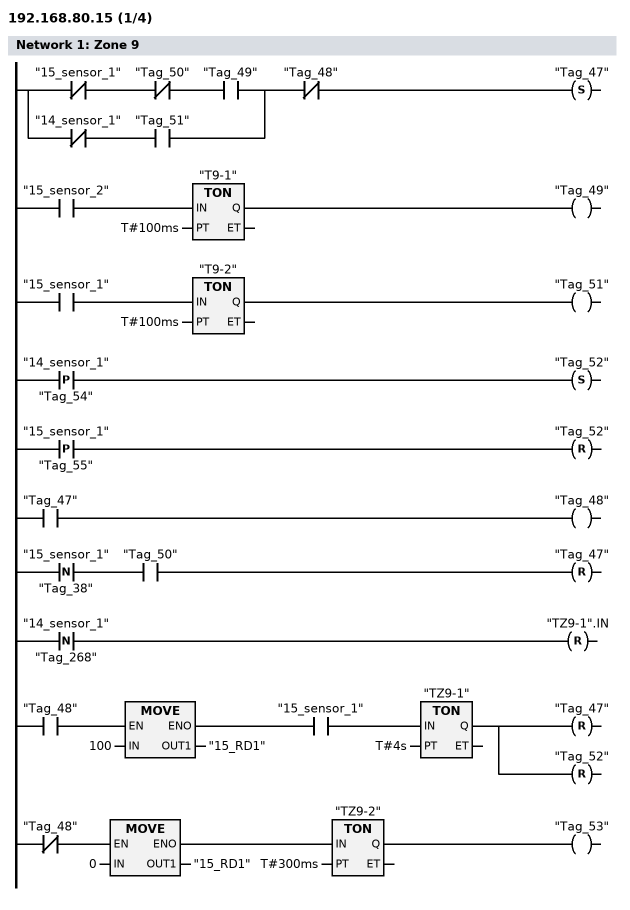
   IF ((NOT "15_sensor_1" AND NOT "Tag_50" AND "Tag_49") OR (NOT "14_sensor_1" AND "Tag_51")) AND NOT "Tag_48" THEN
       "Tag_47" := TRUE;
   END_IF;
   "T9-1".TON(IN := "15_sensor_2", PT := T#100ms);
   "Tag_49" := "T9-1".Q;
   "T9-2".TON(IN := "15_sensor_1", PT := T#100ms);
   "Tag_51" := "T9-2".Q;
   #_w1 := "14_sensor_1" AND NOT "Tag_54";   // rising edge of "14_sensor_1"
   "Tag_54" := "14_sensor_1";
   IF #_w1 THEN "Tag_52" := TRUE; END_IF;
   #_w2 := "15_sensor_1" AND NOT "Tag_55";   // rising edge of "15_sensor_1"
   "Tag_55" := "15_sensor_1";
   IF #_w2 THEN "Tag_52" := FALSE; END_IF;
   "Tag_48" := "Tag_47";
   #_w3 := NOT "15_sensor_1" AND "Tag_38";   // falling edge of "15_sensor_1"
   "Tag_38" := "15_sensor_1";
   IF #_w3 AND "Tag_50" THEN "Tag_47" := FALSE; END_IF;
   #_w4 := NOT "14_sensor_1" AND "Tag_268";   // falling edge of "14_sensor_1"
   "Tag_268" := "14_sensor_1";
   IF #_w4 THEN "TZ9-1".IN := FALSE; END_IF;
   IF "Tag_48" THEN "15_RD1" := 100; END_IF;
   "TZ9-1".TON(IN := "Tag_48" AND "15_sensor_1", PT := T#4s);
   IF "TZ9-1".Q THEN
       "Tag_47" := FALSE;
       "Tag_52" := FALSE;
   END_IF;
   IF NOT "Tag_48" THEN "15_RD1" := 0; END_IF;
   "TZ9-2".TON(IN := NOT "Tag_48", PT := T#300ms);
   "Tag_53" := "TZ9-2".Q;
END_REGION

REGION Network 2: Zone 10
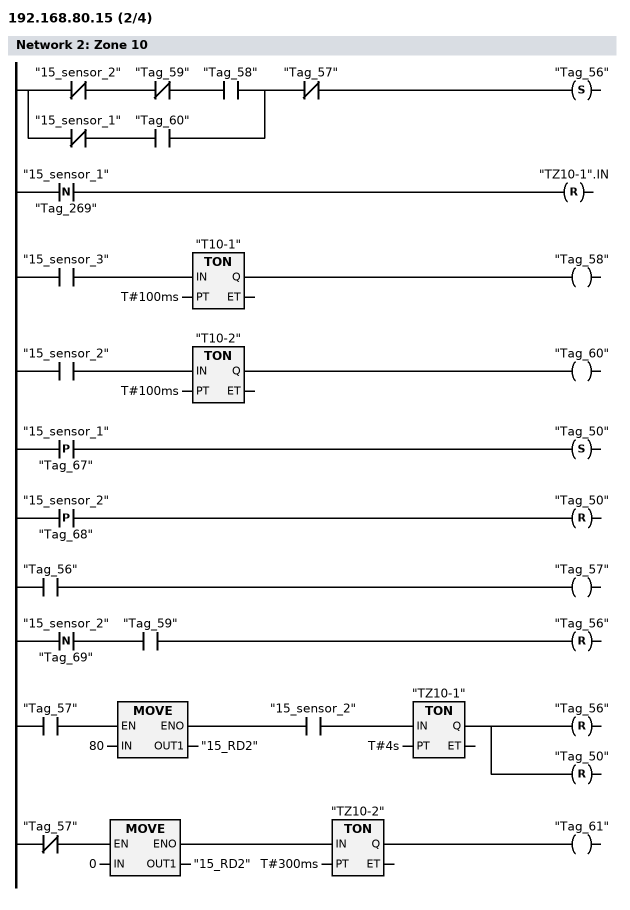
   IF ((NOT "15_sensor_2" AND NOT "Tag_59" AND "Tag_58") OR (NOT "15_sensor_1" AND "Tag_60")) AND NOT "Tag_57" THEN
       "Tag_56" := TRUE;
   END_IF;
   #_w1 := NOT "15_sensor_1" AND "Tag_269";   // falling edge of "15_sensor_1"
   "Tag_269" := "15_sensor_1";
   IF #_w1 THEN "TZ10-1".IN := FALSE; END_IF;
   "T10-1".TON(IN := "15_sensor_3", PT := T#100ms);
   "Tag_58" := "T10-1".Q;
   "T10-2".TON(IN := "15_sensor_2", PT := T#100ms);
   "Tag_60" := "T10-2".Q;
   #_w2 := "15_sensor_1" AND NOT "Tag_67";   // rising edge of "15_sensor_1"
   "Tag_67" := "15_sensor_1";
   IF #_w2 THEN "Tag_50" := TRUE; END_IF;
   #_w3 := "15_sensor_2" AND NOT "Tag_68";   // rising edge of "15_sensor_2"
   "Tag_68" := "15_sensor_2";
   IF #_w3 THEN "Tag_50" := FALSE; END_IF;
   "Tag_57" := "Tag_56";
   #_w4 := NOT "15_sensor_2" AND "Tag_69";   // falling edge of "15_sensor_2"
   "Tag_69" := "15_sensor_2";
   IF #_w4 AND "Tag_59" THEN "Tag_56" := FALSE; END_IF;
   IF "Tag_57" THEN "15_RD2" := 80; END_IF;
   "TZ10-1".TON(IN := "Tag_57" AND "15_sensor_2", PT := T#4s);
   IF "TZ10-1".Q THEN
       "Tag_56" := FALSE;
       "Tag_50" := FALSE;
   END_IF;
   IF NOT "Tag_57" THEN "15_RD2" := 0; END_IF;
   "TZ10-2".TON(IN := NOT "Tag_57", PT := T#300ms);
   "Tag_61" := "TZ10-2".Q;
END_REGION

REGION Network 3: Zone 11
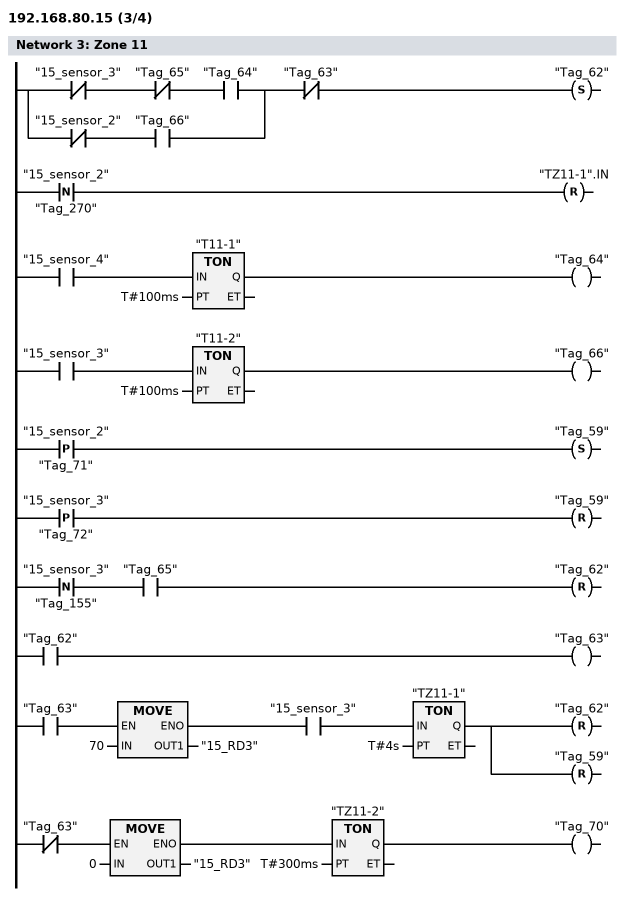
   IF ((NOT "15_sensor_3" AND NOT "Tag_65" AND "Tag_64") OR (NOT "15_sensor_2" AND "Tag_66")) AND NOT "Tag_63" THEN
       "Tag_62" := TRUE;
   END_IF;
   #_w1 := NOT "15_sensor_2" AND "Tag_270";   // falling edge of "15_sensor_2"
   "Tag_270" := "15_sensor_2";
   IF #_w1 THEN "TZ11-1".IN := FALSE; END_IF;
   "T11-1".TON(IN := "15_sensor_4", PT := T#100ms);
   "Tag_64" := "T11-1".Q;
   "T11-2".TON(IN := "15_sensor_3", PT := T#100ms);
   "Tag_66" := "T11-2".Q;
   #_w2 := "15_sensor_2" AND NOT "Tag_71";   // rising edge of "15_sensor_2"
   "Tag_71" := "15_sensor_2";
   IF #_w2 THEN "Tag_59" := TRUE; END_IF;
   #_w3 := "15_sensor_3" AND NOT "Tag_72";   // rising edge of "15_sensor_3"
   "Tag_72" := "15_sensor_3";
   IF #_w3 THEN "Tag_59" := FALSE; END_IF;
   #_w4 := NOT "15_sensor_3" AND "Tag_155";   // falling edge of "15_sensor_3"
   "Tag_155" := "15_sensor_3";
   IF #_w4 AND "Tag_65" THEN "Tag_62" := FALSE; END_IF;
   "Tag_63" := "Tag_62";
   IF "Tag_63" THEN "15_RD3" := 70; END_IF;
   "TZ11-1".TON(IN := "Tag_63" AND "15_sensor_3", PT := T#4s);
   IF "TZ11-1".Q THEN
       "Tag_62" := FALSE;
       "Tag_59" := FALSE;
   END_IF;
   IF NOT "Tag_63" THEN "15_RD3" := 0; END_IF;
   "TZ11-2".TON(IN := NOT "Tag_63", PT := T#300ms);
   "Tag_70" := "TZ11-2".Q;
END_REGION

REGION Network 4: Zone 12
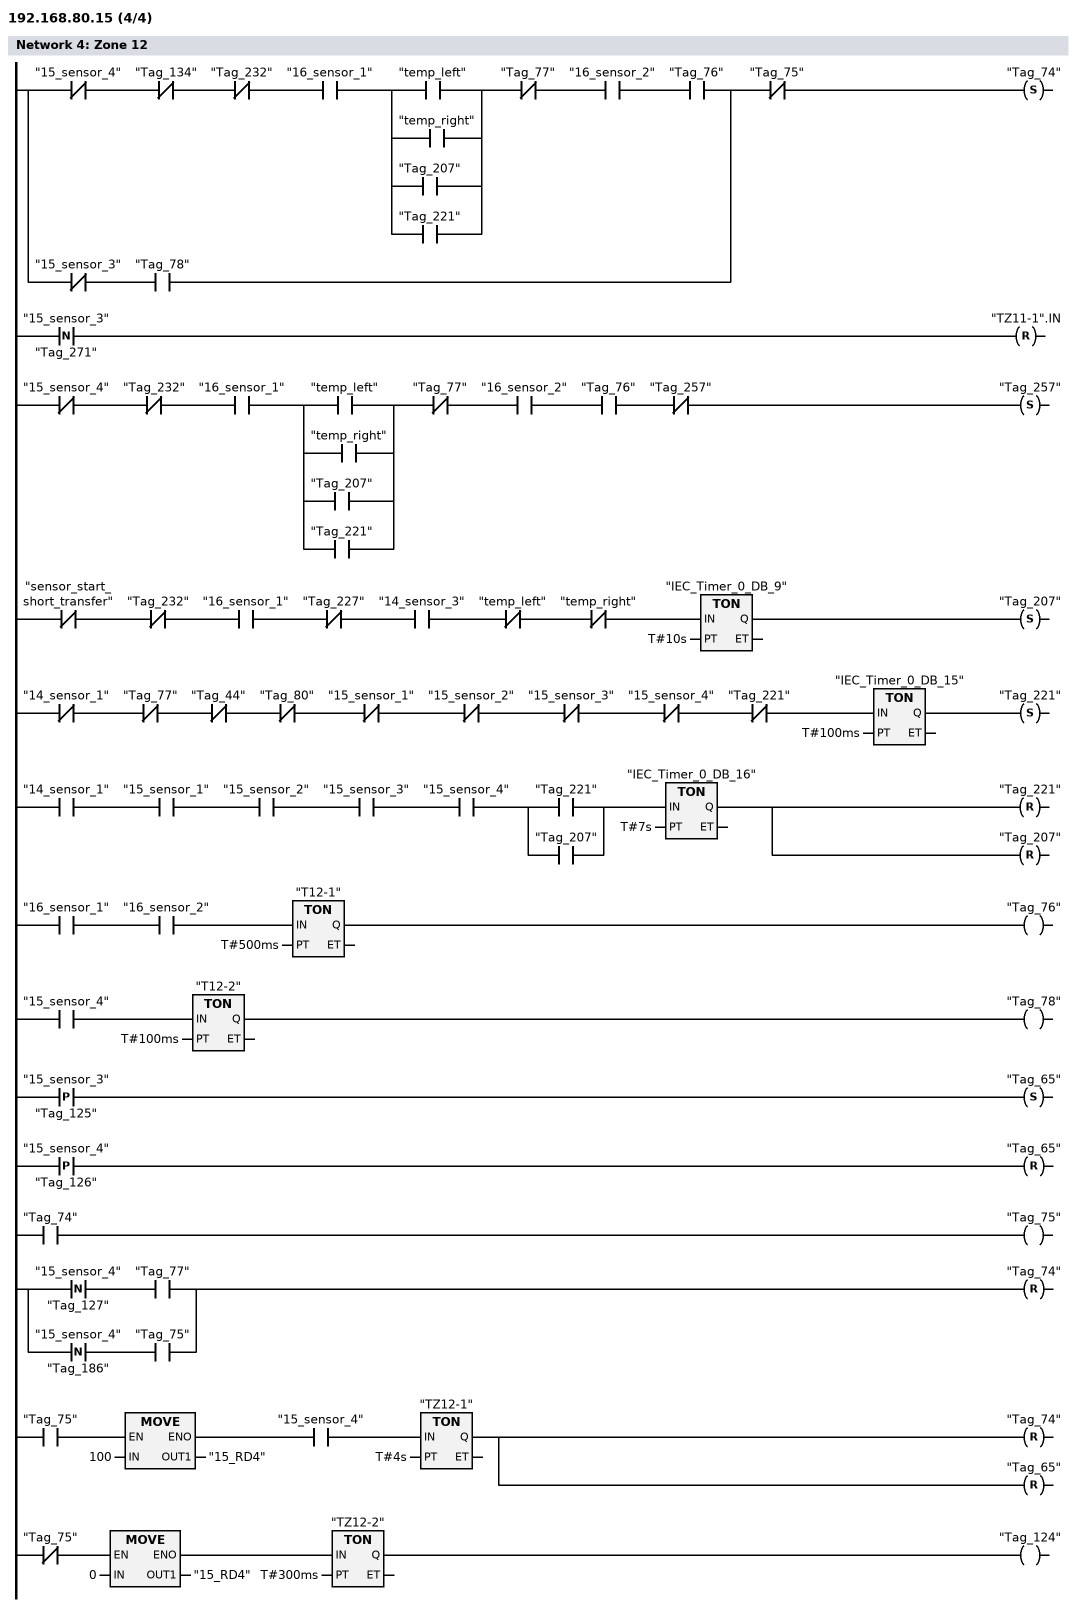
   IF ((NOT "15_sensor_4" AND NOT "Tag_134" AND NOT "Tag_232" AND "16_sensor_1" AND ("temp_left" OR "temp_right" OR "Tag_207" OR "Tag_221") AND NOT "Tag_77" AND "16_sensor_2" AND "Tag_76") OR (NOT "15_sensor_3" AND "Tag_78")) AND NOT "Tag_75" THEN
       "Tag_74" := TRUE;
   END_IF;
   #_w1 := NOT "15_sensor_3" AND "Tag_271";   // falling edge of "15_sensor_3"
   "Tag_271" := "15_sensor_3";
   IF #_w1 THEN "TZ11-1".IN := FALSE; END_IF;
   IF NOT "15_sensor_4" AND NOT "Tag_232" AND "16_sensor_1" AND ("temp_left" OR "temp_right" OR "Tag_207" OR "Tag_221") AND NOT "Tag_77" AND "16_sensor_2" AND "Tag_76" AND NOT "Tag_257" THEN
       "Tag_257" := TRUE;
   END_IF;
   "IEC_Timer_0_DB_9".TON(IN := NOT "sensor_start_short_transfer" AND NOT "Tag_232" AND "16_sensor_1" AND NOT "Tag_227" AND "14_sensor_3" AND NOT "temp_left" AND NOT "temp_right",
                          PT := T#10s);
   IF "IEC_Timer_0_DB_9".Q THEN "Tag_207" := TRUE; END_IF;
   "IEC_Timer_0_DB_15".TON(IN := NOT "14_sensor_1" AND NOT "Tag_77" AND NOT "Tag_44" AND NOT "Tag_80" AND NOT "15_sensor_1" AND NOT "15_sensor_2" AND NOT "15_sensor_3" AND NOT "15_sensor_4" AND NOT "Tag_221",
                           PT := T#100ms);
   IF "IEC_Timer_0_DB_15".Q THEN "Tag_221" := TRUE; END_IF;
   "IEC_Timer_0_DB_16".TON(IN := "14_sensor_1" AND "15_sensor_1" AND "15_sensor_2" AND "15_sensor_3" AND "15_sensor_4" AND ("Tag_221" OR "Tag_207"),
                           PT := T#7s);
   IF "IEC_Timer_0_DB_16".Q THEN
       "Tag_221" := FALSE;
       "Tag_207" := FALSE;
   END_IF;
   "T12-1".TON(IN := "16_sensor_1" AND "16_sensor_2", PT := T#500ms);
   "Tag_76" := "T12-1".Q;
   "T12-2".TON(IN := "15_sensor_4", PT := T#100ms);
   "Tag_78" := "T12-2".Q;
   #_w2 := "15_sensor_3" AND NOT "Tag_125";   // rising edge of "15_sensor_3"
   "Tag_125" := "15_sensor_3";
   IF #_w2 THEN "Tag_65" := TRUE; END_IF;
   #_w3 := "15_sensor_4" AND NOT "Tag_126";   // rising edge of "15_sensor_4"
   "Tag_126" := "15_sensor_4";
   IF #_w3 THEN "Tag_65" := FALSE; END_IF;
   "Tag_75" := "Tag_74";
   #_w4 := NOT "15_sensor_4" AND "Tag_127";   // falling edge of "15_sensor_4"
   "Tag_127" := "15_sensor_4";
   #_w5 := NOT "15_sensor_4" AND "Tag_186";   // falling edge of "15_sensor_4"
   "Tag_186" := "15_sensor_4";
   IF (#_w4 AND "Tag_77") OR (#_w5 AND "Tag_75") THEN "Tag_74" := FALSE; END_IF;
   IF "Tag_75" THEN "15_RD4" := 100; END_IF;
   "TZ12-1".TON(IN := "Tag_75" AND "15_sensor_4", PT := T#4s);
   IF "TZ12-1".Q THEN
       "Tag_74" := FALSE;
       "Tag_65" := FALSE;
   END_IF;
   IF NOT "Tag_75" THEN "15_RD4" := 0; END_IF;
   "TZ12-2".TON(IN := NOT "Tag_75", PT := T#300ms);
   "Tag_124" := "TZ12-2".Q;
END_REGION
END_FUNCTION

FUNCTION "192.168.80.16" : Void   // FC6, LAD
{ S7_Optimized_Access := 'TRUE' }
VERSION : 0.1
   VAR_TEMP   // added for the SCL form of the ladder/FBD networks
      _w1 : Bool;
      _w2 : Bool;
      _w3 : Bool;
      _w4 : Bool;
      _w5 : Bool;
      _w6 : Bool;
      _w7 : Bool;
      _w8 : Bool;
   END_VAR
BEGIN

REGION Network 1: Zone 13
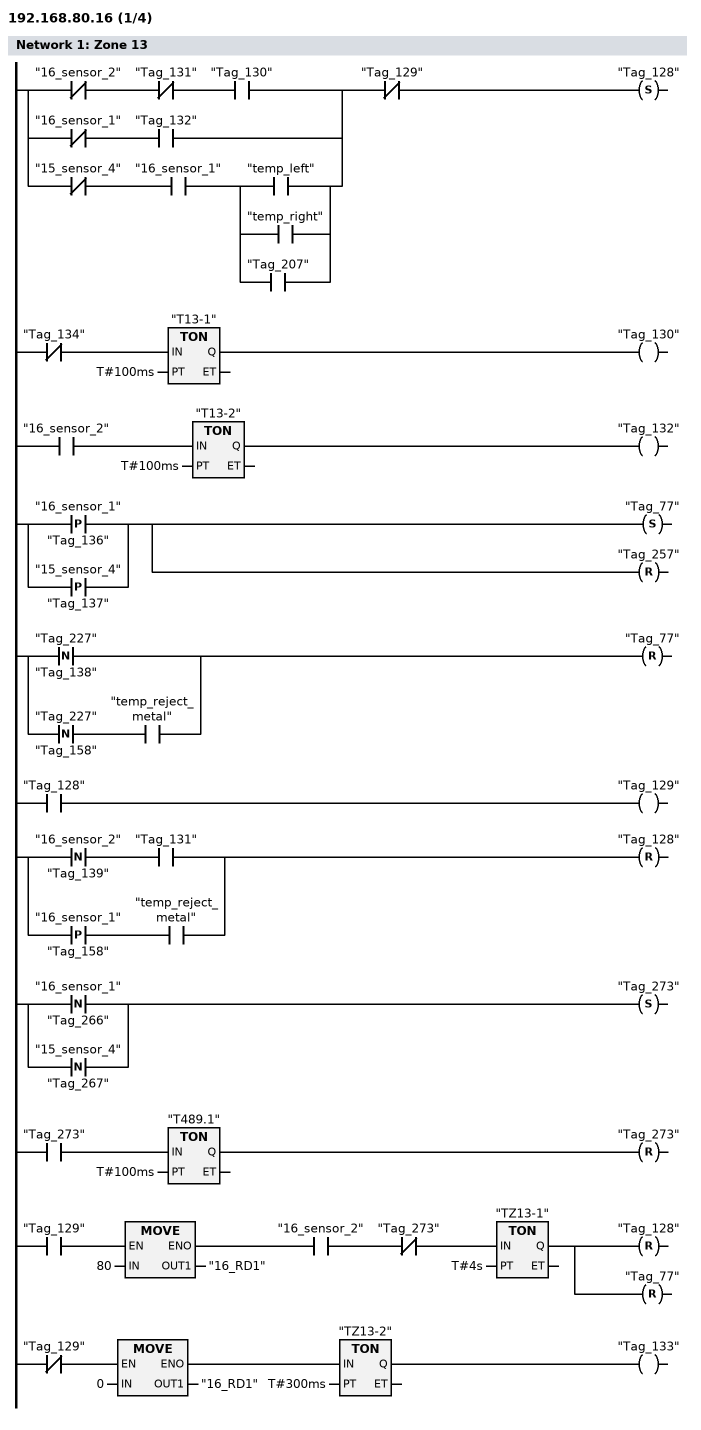
   IF ((NOT "16_sensor_2" AND NOT "Tag_131" AND "Tag_130") OR (NOT "16_sensor_1" AND "Tag_132") OR (NOT "15_sensor_4" AND "16_sensor_1" AND ("temp_left" OR "temp_right" OR "Tag_207"))) AND NOT "Tag_129" THEN
       "Tag_128" := TRUE;
   END_IF;
   "T13-1".TON(IN := NOT "Tag_134", PT := T#100ms);
   "Tag_130" := "T13-1".Q;
   "T13-2".TON(IN := "16_sensor_2", PT := T#100ms);
   "Tag_132" := "T13-2".Q;
   #_w1 := "16_sensor_1" AND NOT "Tag_136";   // rising edge of "16_sensor_1"
   "Tag_136" := "16_sensor_1";
   #_w2 := "15_sensor_4" AND NOT "Tag_137";   // rising edge of "15_sensor_4"
   "Tag_137" := "15_sensor_4";
   IF #_w1 OR #_w2 THEN
       "Tag_77" := TRUE;
       "Tag_257" := FALSE;
   END_IF;
   #_w3 := NOT "Tag_227" AND "Tag_138";   // falling edge of "Tag_227"
   "Tag_138" := "Tag_227";
   #_w4 := NOT "Tag_227" AND "Tag_158";   // falling edge of "Tag_227"
   "Tag_158" := "Tag_227";
   IF #_w3 OR (#_w4 AND "temp_reject_metal") THEN "Tag_77" := FALSE; END_IF;
   "Tag_129" := "Tag_128";
   #_w5 := NOT "16_sensor_2" AND "Tag_139";   // falling edge of "16_sensor_2"
   "Tag_139" := "16_sensor_2";
   #_w6 := "16_sensor_1" AND NOT "Tag_158";   // rising edge of "16_sensor_1"
   "Tag_158" := "16_sensor_1";
   IF (#_w5 AND "Tag_131") OR (#_w6 AND "temp_reject_metal") THEN "Tag_128" := FALSE; END_IF;
   #_w7 := NOT "16_sensor_1" AND "Tag_266";   // falling edge of "16_sensor_1"
   "Tag_266" := "16_sensor_1";
   #_w8 := NOT "15_sensor_4" AND "Tag_267";   // falling edge of "15_sensor_4"
   "Tag_267" := "15_sensor_4";
   IF #_w7 OR #_w8 THEN "Tag_273" := TRUE; END_IF;
   "T489.1".TON(IN := "Tag_273", PT := T#100ms);
   IF "T489.1".Q THEN "Tag_273" := FALSE; END_IF;
   IF "Tag_129" THEN "16_RD1" := 80; END_IF;
   "TZ13-1".TON(IN := "Tag_129" AND "16_sensor_2" AND NOT "Tag_273", PT := T#4s);
   IF "TZ13-1".Q THEN
       "Tag_128" := FALSE;
       "Tag_77" := FALSE;
   END_IF;
   IF NOT "Tag_129" THEN "16_RD1" := 0; END_IF;
   "TZ13-2".TON(IN := NOT "Tag_129", PT := T#300ms);
   "Tag_133" := "TZ13-2".Q;
END_REGION

REGION Network 2: Zone 14
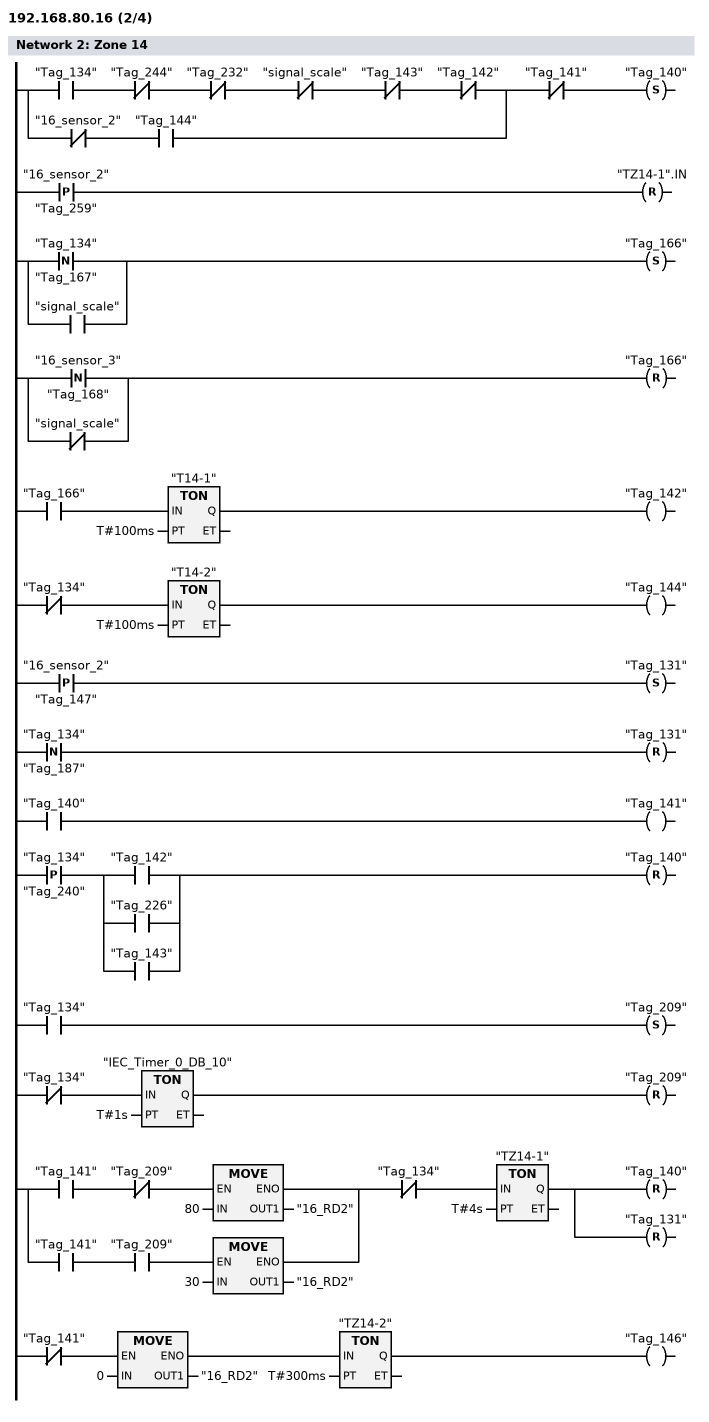
   IF (("Tag_134" AND NOT "Tag_244" AND NOT "Tag_232" AND NOT "signal_scale" AND NOT "Tag_143" AND NOT "Tag_142") OR (NOT "16_sensor_2" AND "Tag_144")) AND NOT "Tag_141" THEN
       "Tag_140" := TRUE;
   END_IF;
   #_w1 := "16_sensor_2" AND NOT "Tag_259";   // rising edge of "16_sensor_2"
   "Tag_259" := "16_sensor_2";
   IF #_w1 THEN "TZ14-1".IN := FALSE; END_IF;
   #_w2 := NOT "Tag_134" AND "Tag_167";   // falling edge of "Tag_134"
   "Tag_167" := "Tag_134";
   IF #_w2 OR "signal_scale" THEN "Tag_166" := TRUE; END_IF;
   #_w3 := NOT "16_sensor_3" AND "Tag_168";   // falling edge of "16_sensor_3"
   "Tag_168" := "16_sensor_3";
   IF #_w3 OR NOT "signal_scale" THEN "Tag_166" := FALSE; END_IF;
   "T14-1".TON(IN := "Tag_166", PT := T#100ms);
   "Tag_142" := "T14-1".Q;
   "T14-2".TON(IN := NOT "Tag_134", PT := T#100ms);
   "Tag_144" := "T14-2".Q;
   #_w4 := "16_sensor_2" AND NOT "Tag_147";   // rising edge of "16_sensor_2"
   "Tag_147" := "16_sensor_2";
   IF #_w4 THEN "Tag_131" := TRUE; END_IF;
   #_w5 := NOT "Tag_134" AND "Tag_187";   // falling edge of "Tag_134"
   "Tag_187" := "Tag_134";
   IF #_w5 THEN "Tag_131" := FALSE; END_IF;
   "Tag_141" := "Tag_140";
   #_w6 := "Tag_134" AND NOT "Tag_240";   // rising edge of "Tag_134"
   "Tag_240" := "Tag_134";
   IF #_w6 AND ("Tag_142" OR "Tag_226" OR "Tag_143") THEN "Tag_140" := FALSE; END_IF;
   IF "Tag_134" THEN "Tag_209" := TRUE; END_IF;
   "IEC_Timer_0_DB_10".TON(IN := NOT "Tag_134", PT := T#1s);
   IF "IEC_Timer_0_DB_10".Q THEN "Tag_209" := FALSE; END_IF;
   #_w7 := "Tag_141" AND NOT "Tag_209";
   IF #_w7 THEN "16_RD2" := 80; END_IF;
   #_w8 := "Tag_141" AND "Tag_209";
   IF #_w8 THEN "16_RD2" := 30; END_IF;
   "TZ14-1".TON(IN := (#_w7 OR #_w8) AND NOT "Tag_134", PT := T#4s);
   IF "TZ14-1".Q THEN
       "Tag_140" := FALSE;
       "Tag_131" := FALSE;
   END_IF;
   IF NOT "Tag_141" THEN "16_RD2" := 0; END_IF;
   "TZ14-2".TON(IN := NOT "Tag_141", PT := T#300ms);
   "Tag_146" := "TZ14-2".Q;
END_REGION

REGION Network 3: Zone 15
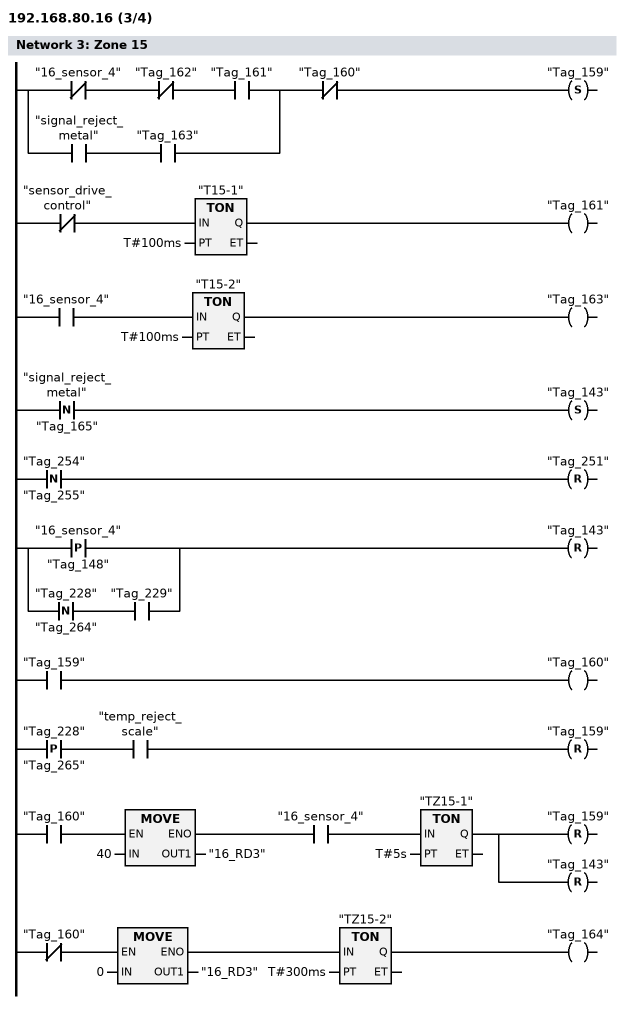
   IF ((NOT "16_sensor_4" AND NOT "Tag_162" AND "Tag_161") OR ("signal_reject_metal" AND "Tag_163")) AND NOT "Tag_160" THEN
       "Tag_159" := TRUE;
   END_IF;
   "T15-1".TON(IN := NOT "sensor_drive_control", PT := T#100ms);
   "Tag_161" := "T15-1".Q;
   "T15-2".TON(IN := "16_sensor_4", PT := T#100ms);
   "Tag_163" := "T15-2".Q;
   #_w1 := NOT "signal_reject_metal" AND "Tag_165";   // falling edge of "signal_reject_metal"
   "Tag_165" := "signal_reject_metal";
   IF #_w1 THEN "Tag_143" := TRUE; END_IF;
   #_w2 := NOT "Tag_254" AND "Tag_255";   // falling edge of "Tag_254"
   "Tag_255" := "Tag_254";
   IF #_w2 THEN "Tag_251" := FALSE; END_IF;
   #_w3 := "16_sensor_4" AND NOT "Tag_148";   // rising edge of "16_sensor_4"
   "Tag_148" := "16_sensor_4";
   #_w4 := NOT "Tag_228" AND "Tag_264";   // falling edge of "Tag_228"
   "Tag_264" := "Tag_228";
   IF #_w3 OR (#_w4 AND "Tag_229") THEN "Tag_143" := FALSE; END_IF;
   "Tag_160" := "Tag_159";
   #_w5 := "Tag_228" AND NOT "Tag_265";   // rising edge of "Tag_228"
   "Tag_265" := "Tag_228";
   IF #_w5 AND "temp_reject_scale" THEN "Tag_159" := FALSE; END_IF;
   IF "Tag_160" THEN "16_RD3" := 40; END_IF;
   "TZ15-1".TON(IN := "Tag_160" AND "16_sensor_4", PT := T#5s);
   IF "TZ15-1".Q THEN
       "Tag_159" := FALSE;
       "Tag_143" := FALSE;
   END_IF;
   IF NOT "Tag_160" THEN "16_RD3" := 0; END_IF;
   "TZ15-2".TON(IN := NOT "Tag_160", PT := T#300ms);
   "Tag_164" := "TZ15-2".Q;
END_REGION

REGION Network 4: Zone 16
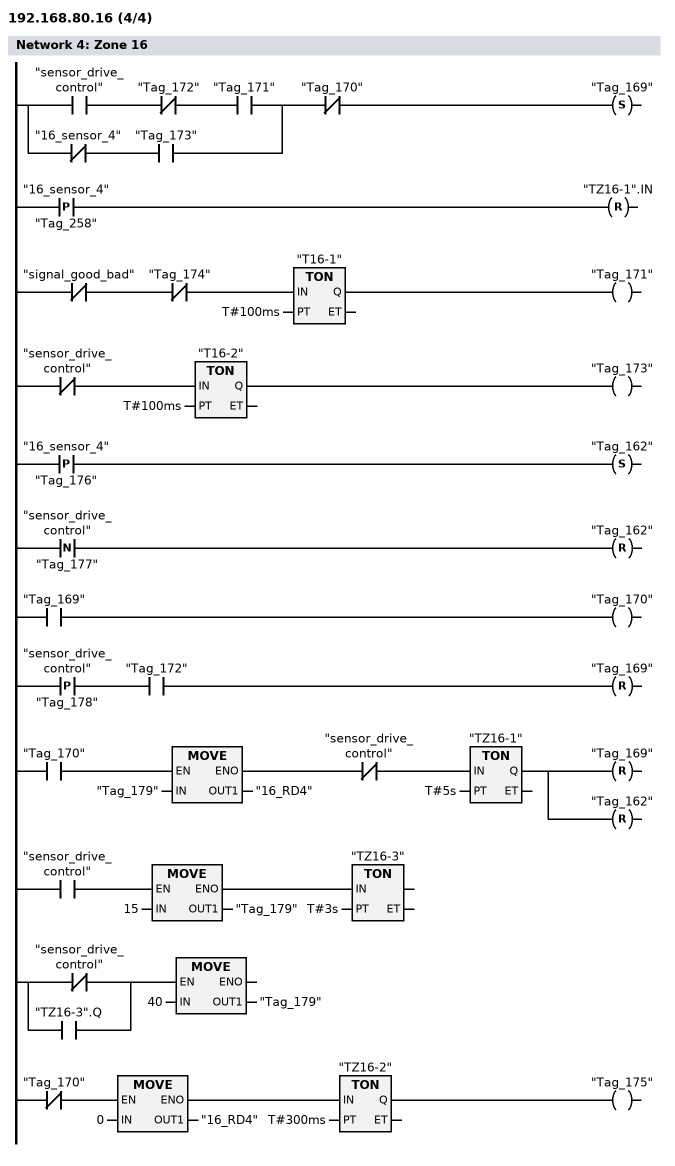
   IF (("sensor_drive_control" AND NOT "Tag_172" AND "Tag_171") OR (NOT "16_sensor_4" AND "Tag_173")) AND NOT "Tag_170" THEN
       "Tag_169" := TRUE;
   END_IF;
   #_w1 := "16_sensor_4" AND NOT "Tag_258";   // rising edge of "16_sensor_4"
   "Tag_258" := "16_sensor_4";
   IF #_w1 THEN "TZ16-1".IN := FALSE; END_IF;
   "T16-1".TON(IN := NOT "signal_good_bad" AND NOT "Tag_174", PT := T#100ms);
   "Tag_171" := "T16-1".Q;
   "T16-2".TON(IN := NOT "sensor_drive_control", PT := T#100ms);
   "Tag_173" := "T16-2".Q;
   #_w2 := "16_sensor_4" AND NOT "Tag_176";   // rising edge of "16_sensor_4"
   "Tag_176" := "16_sensor_4";
   IF #_w2 THEN "Tag_162" := TRUE; END_IF;
   #_w3 := NOT "sensor_drive_control" AND "Tag_177";   // falling edge of "sensor_drive_control"
   "Tag_177" := "sensor_drive_control";
   IF #_w3 THEN "Tag_162" := FALSE; END_IF;
   "Tag_170" := "Tag_169";
   #_w4 := "sensor_drive_control" AND NOT "Tag_178";   // rising edge of "sensor_drive_control"
   "Tag_178" := "sensor_drive_control";
   IF #_w4 AND "Tag_172" THEN "Tag_169" := FALSE; END_IF;
   IF "Tag_170" THEN "16_RD4" := "Tag_179"; END_IF;
   "TZ16-1".TON(IN := "Tag_170" AND NOT "sensor_drive_control", PT := T#5s);
   IF "TZ16-1".Q THEN
       "Tag_169" := FALSE;
       "Tag_162" := FALSE;
   END_IF;
   IF "sensor_drive_control" THEN "Tag_179" := 15; END_IF;
   "TZ16-3".TON(IN := "sensor_drive_control", PT := T#3s);
   IF NOT "sensor_drive_control" OR "TZ16-3".Q THEN "Tag_179" := 40; END_IF;
   IF NOT "Tag_170" THEN "16_RD4" := 0; END_IF;
   "TZ16-2".TON(IN := NOT "Tag_170", PT := T#300ms);
   "Tag_175" := "TZ16-2".Q;
END_REGION
END_FUNCTION

FUNCTION "drive_control" : Void   // FC7, LAD
{ S7_Optimized_Access := 'TRUE' }
VERSION : 0.1
   VAR_TEMP   // added for the SCL form of the ladder/FBD networks
      _w1 : Bool;
      _w2 : Bool;
      _w3 : Bool;
      _w4 : Bool;
      _w5 : Bool;
   END_VAR
BEGIN

REGION Network 1
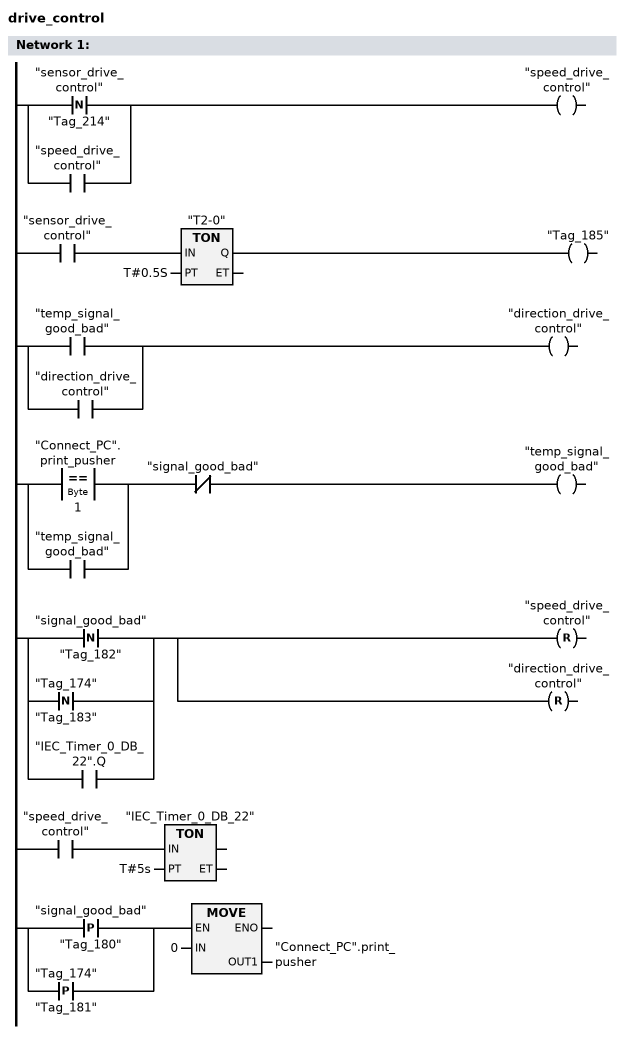
   #_w1 := NOT "sensor_drive_control" AND "Tag_214";   // falling edge of "sensor_drive_control"
   "Tag_214" := "sensor_drive_control";
   "speed_drive_control" := #_w1 OR "speed_drive_control";
   "T2-0".TON(IN := "sensor_drive_control", PT := T#0.5S);
   "Tag_185" := "T2-0".Q;
   "direction_drive_control" := "temp_signal_good_bad" OR "direction_drive_control";
   "temp_signal_good_bad" := (("Connect_PC".print_pusher = 1) OR "temp_signal_good_bad") AND NOT "signal_good_bad";
   #_w2 := NOT "signal_good_bad" AND "Tag_182";   // falling edge of "signal_good_bad"
   "Tag_182" := "signal_good_bad";
   #_w3 := NOT "Tag_174" AND "Tag_183";   // falling edge of "Tag_174"
   "Tag_183" := "Tag_174";
   IF #_w2 OR #_w3 OR "IEC_Timer_0_DB_22".Q THEN
       "speed_drive_control" := FALSE;
       "direction_drive_control" := FALSE;
   END_IF;
   "IEC_Timer_0_DB_22".TON(IN := "speed_drive_control", PT := T#5s);
   #_w4 := "signal_good_bad" AND NOT "Tag_180";   // rising edge of "signal_good_bad"
   "Tag_180" := "signal_good_bad";
   #_w5 := "Tag_174" AND NOT "Tag_181";   // rising edge of "Tag_174"
   "Tag_181" := "Tag_174";
   IF #_w4 OR #_w5 THEN "Connect_PC".print_pusher := 0; END_IF;
END_REGION
END_FUNCTION

ORGANIZATION_BLOCK "Main"   // OB1, LAD, ProgramCycle
TITLE = "Main Program Sweep (Cycle)"
{ S7_Optimized_Access := 'TRUE' }
VERSION : 0.1
   VAR_INPUT
      Initial_Call : Bool;   // Initial call of this OB
      Remanence : Bool;   // =True, if remanent data are available
   END_VAR
   VAR_TEMP   // added for the SCL form of the ladder/FBD networks
      _w1 : Bool;
      _w2 : Bool;
   END_VAR
BEGIN

REGION Network 1
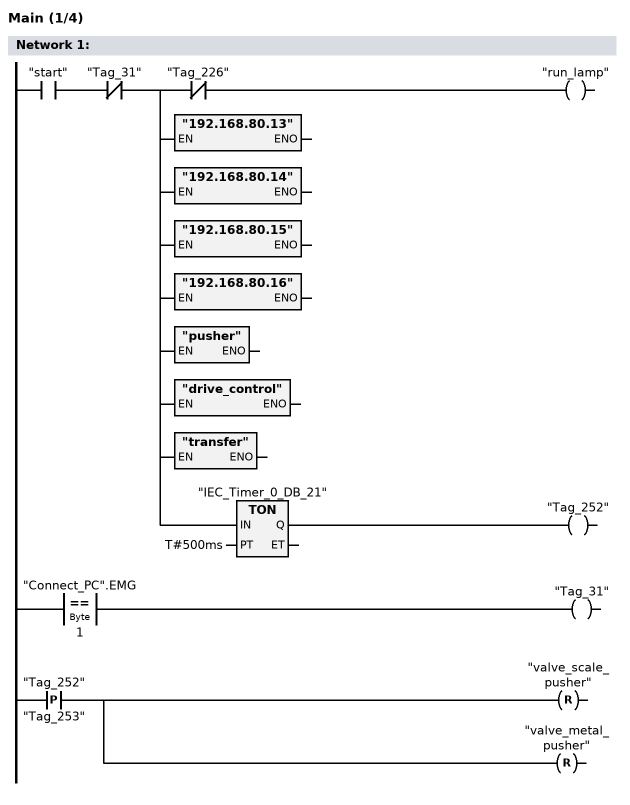
   #_w1 := "start" AND NOT "Tag_31";
   "run_lamp" := #_w1 AND NOT "Tag_226";
   IF #_w1 THEN
       "192.168.80.13"();
       "192.168.80.14"();
       "192.168.80.15"();
       "192.168.80.16"();
       "pusher"();
       "drive_control"();
       "transfer"();
   END_IF;
   "IEC_Timer_0_DB_21".TON(IN := #_w1, PT := T#500ms);
   "Tag_252" := "IEC_Timer_0_DB_21".Q;
   "Tag_31" := "Connect_PC".EMG = 1;
   #_w2 := "Tag_252" AND NOT "Tag_253";   // rising edge of "Tag_252"
   "Tag_253" := "Tag_252";
   IF #_w2 THEN
       "valve_scale_pusher" := FALSE;
       "valve_metal_pusher" := FALSE;
   END_IF;
END_REGION

REGION Network 2
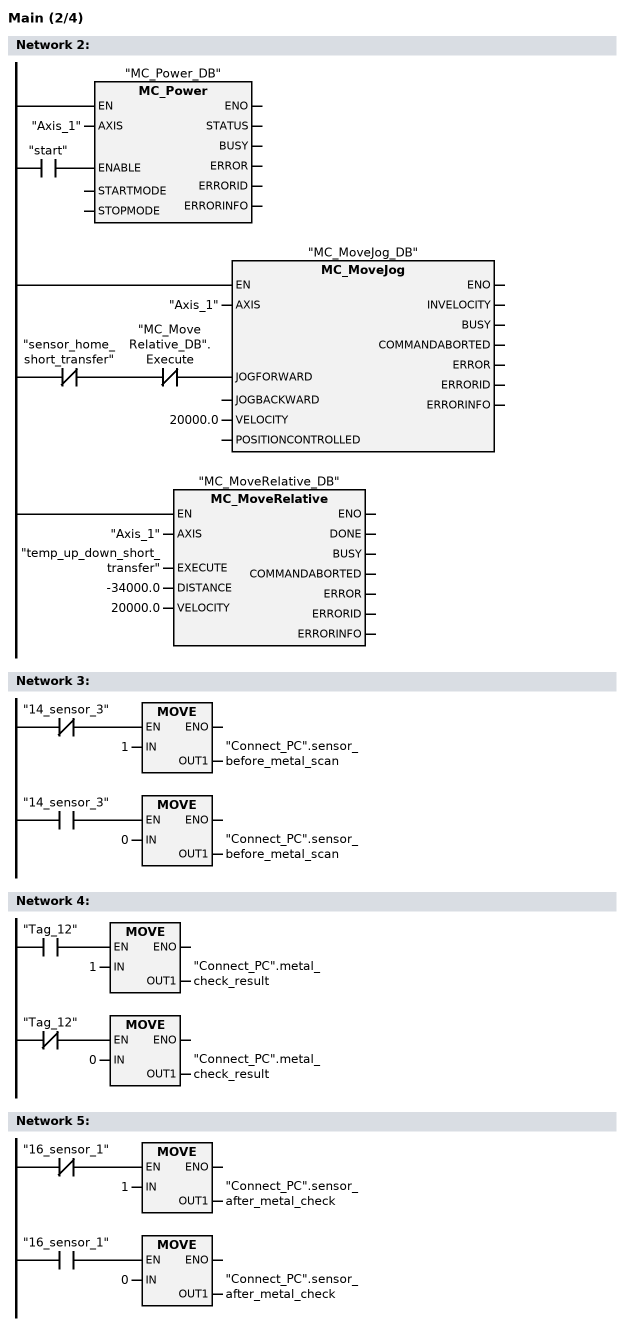
   "MC_Power_DB"(Axis := "Axis_1", Enable := "start");   // MC_Power
   "MC_MoveJog_DB"(Axis := "Axis_1",   // MC_MoveJog
                   JogForward := NOT "sensor_home_short_transfer" AND NOT "MC_MoveRelative_DB".Execute,
                   Velocity := 20000.0);
   "MC_MoveRelative_DB"(Axis := "Axis_1",   // MC_MoveRelative
                        Execute := "temp_up_down_short_transfer",
                        Distance := -34000.0,
                        Velocity := 20000.0);
END_REGION

REGION Network 3
   RUNG wire#powerrail
      I_Contact( "14_sensor_3" )
      Move(in := 1, out1 => "Connect_PC".sensor_before_metal_scan)
   END_RUNG
   RUNG wire#powerrail
      Contact( "14_sensor_3" )
      Move(in := 0, out1 => "Connect_PC".sensor_before_metal_scan)
   END_RUNG
   // the same network as SCL:
   IF NOT "14_sensor_3" THEN "Connect_PC".sensor_before_metal_scan := 1; END_IF;
   IF "14_sensor_3" THEN "Connect_PC".sensor_before_metal_scan := 0; END_IF;
END_REGION

REGION Network 4
   RUNG wire#powerrail
      Contact( "Tag_12" )
      Move(in := 1, out1 => "Connect_PC".metal_check_result)
   END_RUNG
   RUNG wire#powerrail
      I_Contact( "Tag_12" )
      Move(in := 0, out1 => "Connect_PC".metal_check_result)
   END_RUNG
   // the same network as SCL:
   IF "Tag_12" THEN "Connect_PC".metal_check_result := 1; END_IF;
   IF NOT "Tag_12" THEN "Connect_PC".metal_check_result := 0; END_IF;
END_REGION

REGION Network 5
   RUNG wire#powerrail
      I_Contact( "16_sensor_1" )
      Move(in := 1, out1 => "Connect_PC".sensor_after_metal_check)
   END_RUNG
   RUNG wire#powerrail
      Contact( "16_sensor_1" )
      Move(in := 0, out1 => "Connect_PC".sensor_after_metal_check)
   END_RUNG
   // the same network as SCL:
   IF NOT "16_sensor_1" THEN "Connect_PC".sensor_after_metal_check := 1; END_IF;
   IF "16_sensor_1" THEN "Connect_PC".sensor_after_metal_check := 0; END_IF;
END_REGION

REGION Network 6
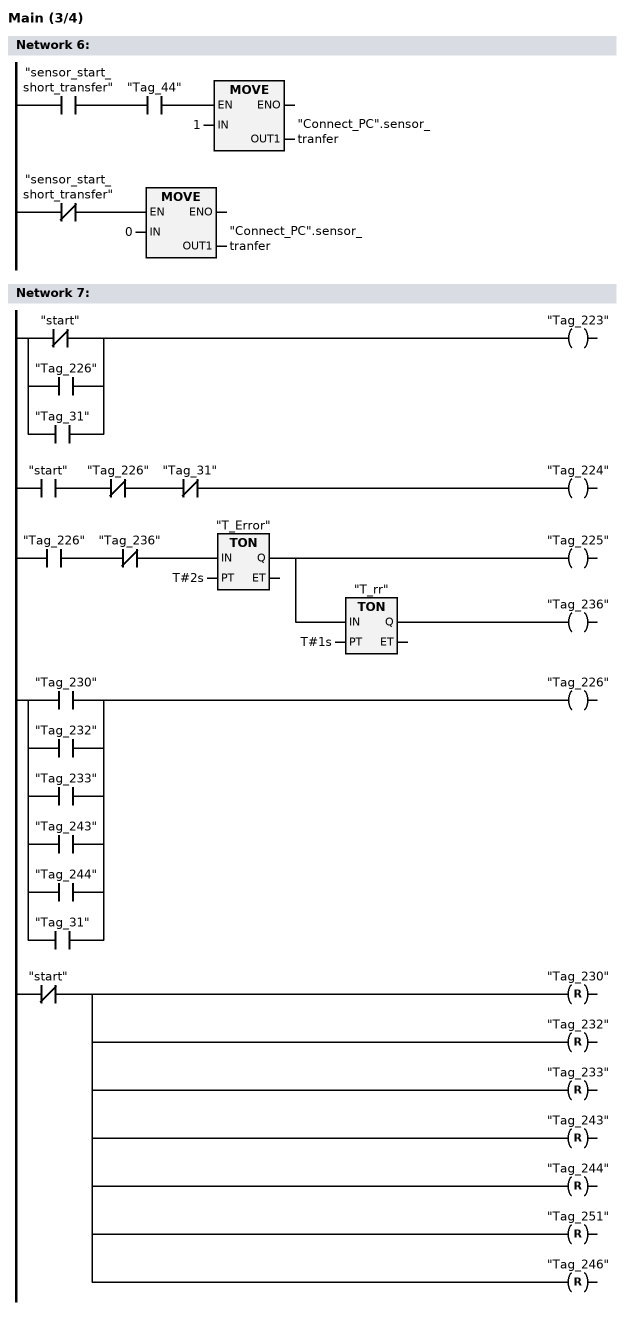
   RUNG wire#powerrail
      Contact( "sensor_start_short_transfer" )
      Contact( "Tag_44" )
      Move(in := 1, out1 => "Connect_PC".sensor_tranfer)
   END_RUNG
   RUNG wire#powerrail
      I_Contact( "sensor_start_short_transfer" )
      Move(in := 0, out1 => "Connect_PC".sensor_tranfer)
   END_RUNG
   // the same network as SCL:
   IF "sensor_start_short_transfer" AND "Tag_44" THEN "Connect_PC".sensor_tranfer := 1; END_IF;
   IF NOT "sensor_start_short_transfer" THEN "Connect_PC".sensor_tranfer := 0; END_IF;
END_REGION

REGION Network 7
   "Tag_223" := NOT "start" OR "Tag_226" OR "Tag_31";
   "Tag_224" := "start" AND NOT "Tag_226" AND NOT "Tag_31";
   "T_Error".TON(IN := "Tag_226" AND NOT "Tag_236", PT := T#2s);
   "Tag_225" := "T_Error".Q;
   "T_rr".TON(IN := "T_Error".Q, PT := T#1s);
   "Tag_236" := "T_rr".Q;
   "Tag_226" := "Tag_230" OR "Tag_232" OR "Tag_233" OR "Tag_243" OR "Tag_244" OR "Tag_31";
   IF NOT "start" THEN
       "Tag_230" := FALSE;
       "Tag_232" := FALSE;
       "Tag_233" := FALSE;
       "Tag_243" := FALSE;
       "Tag_244" := FALSE;
       "Tag_251" := FALSE;
       "Tag_246" := FALSE;
   END_IF;
END_REGION

REGION Network 8
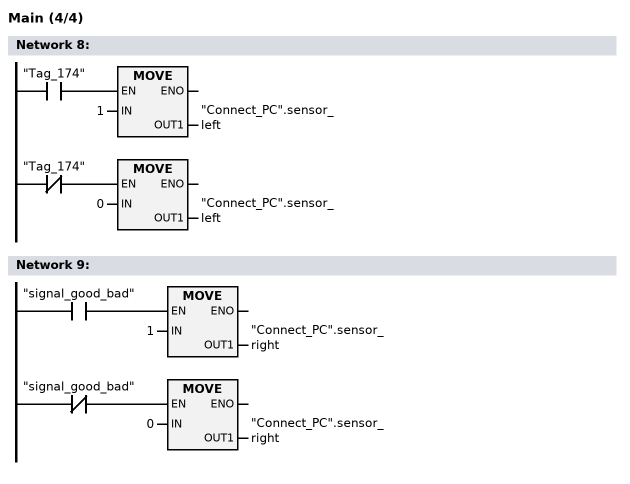
   RUNG wire#powerrail
      Contact( "Tag_174" )
      Move(in := 1, out1 => "Connect_PC".sensor_left)
   END_RUNG
   RUNG wire#powerrail
      I_Contact( "Tag_174" )
      Move(in := 0, out1 => "Connect_PC".sensor_left)
   END_RUNG
   // the same network as SCL:
   IF "Tag_174" THEN "Connect_PC".sensor_left := 1; END_IF;
   IF NOT "Tag_174" THEN "Connect_PC".sensor_left := 0; END_IF;
END_REGION

REGION Network 9
   RUNG wire#powerrail
      Contact( "signal_good_bad" )
      Move(in := 1, out1 => "Connect_PC".sensor_right)
   END_RUNG
   RUNG wire#powerrail
      I_Contact( "signal_good_bad" )
      Move(in := 0, out1 => "Connect_PC".sensor_right)
   END_RUNG
   // the same network as SCL:
   IF "signal_good_bad" THEN "Connect_PC".sensor_right := 1; END_IF;
   IF NOT "signal_good_bad" THEN "Connect_PC".sensor_right := 0; END_IF;
END_REGION
END_ORGANIZATION_BLOCK